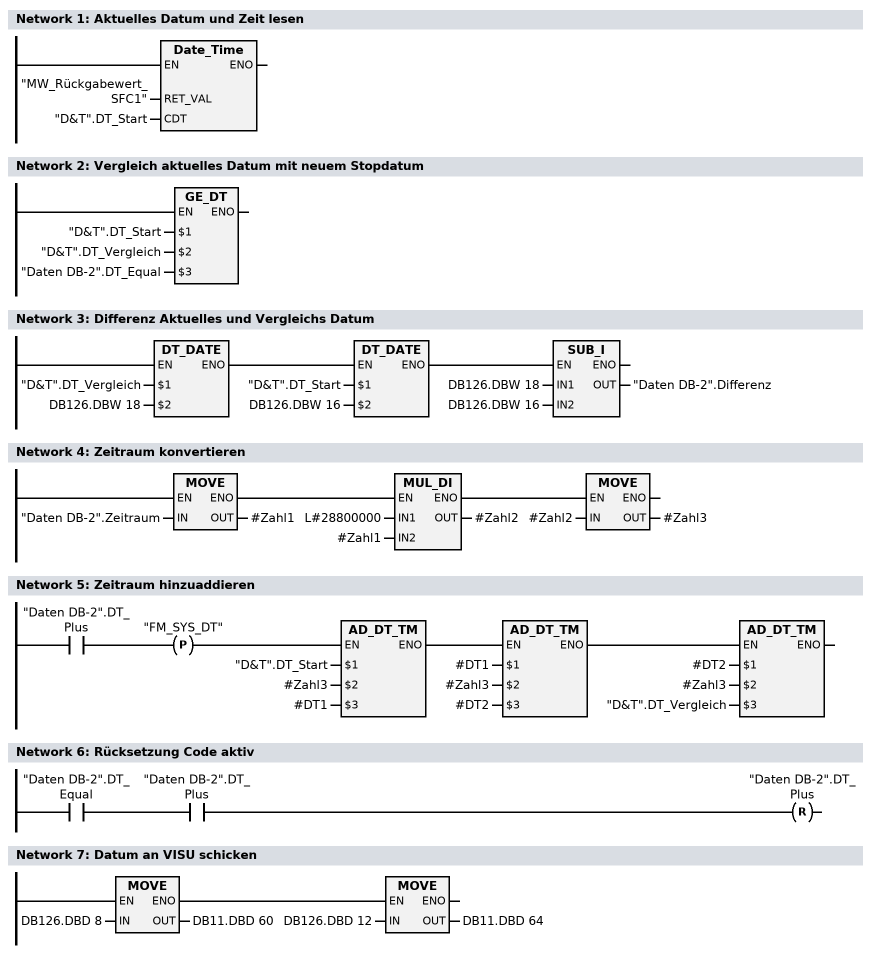
NETWORK
TITLE = Aktuelles Datum und Zeit lesen
      CALL  "Date_Time" (
           RET_VAL                  := "MW_Rückgabewert_SFC1",
           CDT                      := "D&T".DT_Start);
NETWORK
TITLE = Vergleich aktuelles Datum mit neuem Stopdatum
      CALL  "GE_DT" (
           $1                       := "D&T".DT_Start,
           $2                       := "D&T".DT_Vergleich,
           $3                       := "Daten DB-2".DT_Equal);
      NOP   0;
NETWORK
TITLE = Differenz Aktuelles und Vergleichs Datum
      A(;
      A(;
      CALL  "DT_DATE" (
           $1                       := "D&T".DT_Vergleich,
           $2                       := DB126.DBW 18);
      A     BR;
      );
      JNB   _001;
      CALL  "DT_DATE" (
           $1                       := "D&T".DT_Start,
           $2                       := DB126.DBW 16);
_001: A     BR;
      );
      JNB   _002;
      L     DB126.DBW 18;
      L     DB126.DBW 16;
      -I;
      T     "Daten DB-2".Differenz;
_002: NOP   0;
NETWORK
TITLE = Zeitraum konvertieren
      A(;
      A(;
      L     "Daten DB-2".Zeitraum;
      T     #Zahl1;
      SET;
      SAVE;
      CLR;
      A     BR;
      );
      JNB   _003;
      L     L#28800000;
      L     #Zahl1;
      *D;
      T     #Zahl2;
      AN    OV;
      SAVE;
      CLR;
_003: A     BR;
      );
      JNB   _004;
      L     #Zahl2;
      T     #Zahl3;
_004: NOP   0;
NETWORK
TITLE = Zeitraum hinzuaddieren
      A(;
      A(;
      A     "Daten DB-2".DT_Plus;
      FP    "FM_SYS_DT";
      JNB   _005;
      CALL  "AD_DT_TM" (
           $1                       := "D&T".DT_Start,
           $2                       := #Zahl3,
           $3                       := #DT1);
_005: A     BR;
      );
      JNB   _006;
      CALL  "AD_DT_TM" (
           $1                       := #DT1,
           $2                       := #Zahl3,
           $3                       := #DT2);
_006: A     BR;
      );
      JNB   _007;
      CALL  "AD_DT_TM" (
           $1                       := #DT2,
           $2                       := #Zahl3,
           $3                       := "D&T".DT_Vergleich);
_007: NOP   0;
NETWORK
TITLE = Rücksetzung Code aktiv
      A     "Daten DB-2".DT_Equal;
      A     "Daten DB-2".DT_Plus;
      R     "Daten DB-2".DT_Plus;
NETWORK
TITLE = Datum an VISU schicken
      A(;
      L     DB126.DBD 8;
      T     DB11.DBD 60;
      SET;
      SAVE;
      CLR;
      A     BR;
      );
      JNB   _008;
      L     DB126.DBD 12;
      T     DB11.DBD 64;
_008: NOP   0;
END_FUNCTION

// FC 127: know-how protected block, not included

// FC 128: know-how protected block, not included

// FC 129: know-how protected block, not included

// FC 130: know-how protected block, not included

FUNCTION "CutterSpeed-A4VG250" : VOID	// FC 140
TITLE = Volumenstromeinstellung für Schürfrad BKAG132kW/CSG355
AUTHOR : Simdon
FAMILY : Cutter
NAME : CutVol3
VERSION : 0.1
VAR_TEMP
  Ltr_200 : BOOL ;	//115 ltr/min
  Ltr_270 : BOOL ;	//270 ltr/min
  Ltr_max : BOOL ;	//max. Fördermenge
END_VAR
BEGIN
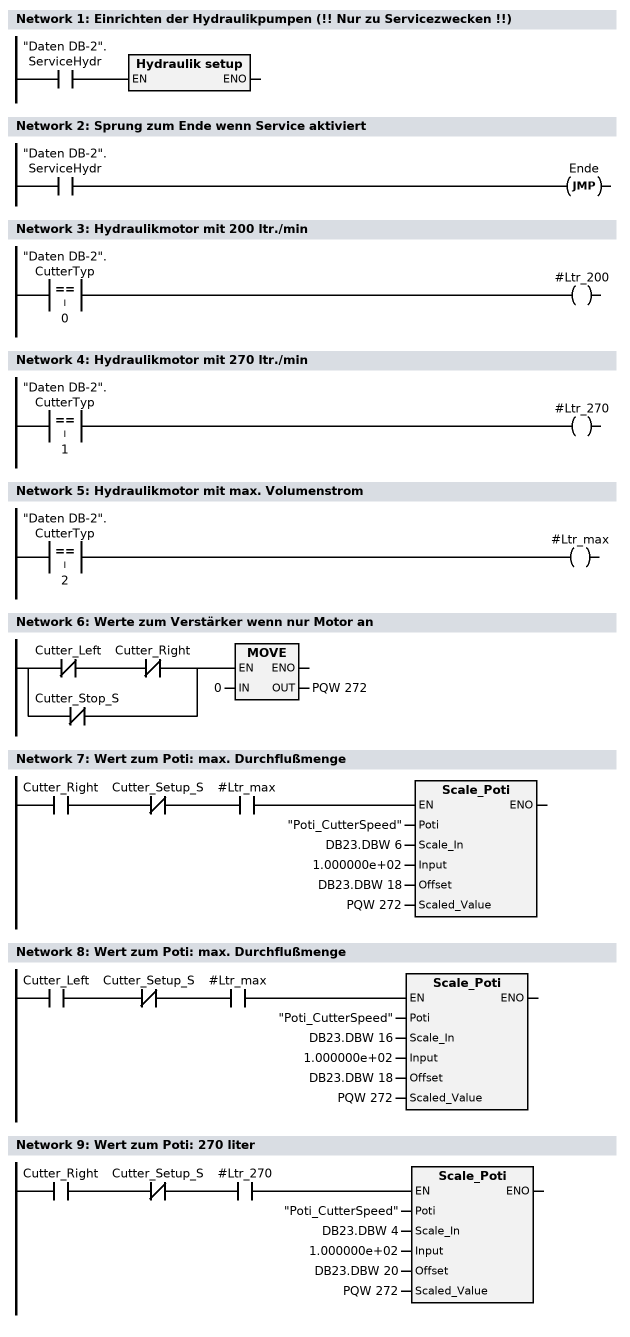
NETWORK
TITLE = Einrichten der Hydraulikpumpen (!! Nur zu Servicezwecken !!)
      A     "Daten DB-2".ServiceHydr;
      JNB   _001;
      CALL  "Hydraulik setup";
_001: NOP   0;
NETWORK
TITLE = Sprung zum Ende wenn Service aktiviert
      A     "Daten DB-2".ServiceHydr;
      JC    Ende;
NETWORK
TITLE = Hydraulikmotor mit 200 ltr./min
      L     "Daten DB-2".CutterTyp;
      L     0;
      ==I;
      =     #Ltr_200;
NETWORK
TITLE = Hydraulikmotor mit 270 ltr./min
      L     "Daten DB-2".CutterTyp;
      L     1;
      ==I;
      =     #Ltr_270;
NETWORK
TITLE = Hydraulikmotor mit max. Volumenstrom
      L     "Daten DB-2".CutterTyp;
      L     2;
      ==I;
      =     #Ltr_max;
NETWORK
TITLE = Werte zum Verstärker wenn nur Motor an
      A(;
      AN    "Cutter_Left";
      AN    "Cutter_Right";
      ON    "Cutter_Stop_S";
      );
      JNB   _002;
      L     0;
      T     PQW 272;
_002: NOP   0;
NETWORK
TITLE = Wert zum Poti: max. Durchflußmenge
      A     "Cutter_Right";
      AN    "Cutter_Setup_S";
      A     #Ltr_max;
      JNB   _003;
      CALL  "Scale_Poti" (
           Poti                     := "Poti_CutterSpeed",
           Scale_In                 := DB23.DBW 6,
           Input                    := 1.000000e+02,
           Offset                   := DB23.DBW 18,
           Scaled_Value             := PQW 272);
_003: NOP   0;
NETWORK
TITLE = Wert zum Poti: max. Durchflußmenge
      A     "Cutter_Left";
      AN    "Cutter_Setup_S";
      A     #Ltr_max;
      JNB   _004;
      CALL  "Scale_Poti" (
           Poti                     := "Poti_CutterSpeed",
           Scale_In                 := DB23.DBW 16,
           Input                    := 1.000000e+02,
           Offset                   := DB23.DBW 18,
           Scaled_Value             := PQW 272);
_004: NOP   0;
NETWORK
TITLE = Wert zum Poti: 270 liter
      A     "Cutter_Right";
      AN    "Cutter_Setup_S";
      A     #Ltr_270;
      JNB   _005;
      CALL  "Scale_Poti" (
           Poti                     := "Poti_CutterSpeed",
           Scale_In                 := DB23.DBW 4,
           Input                    := 1.000000e+02,
           Offset                   := DB23.DBW 20,
           Scaled_Value             := PQW 272);
_005: NOP   0;
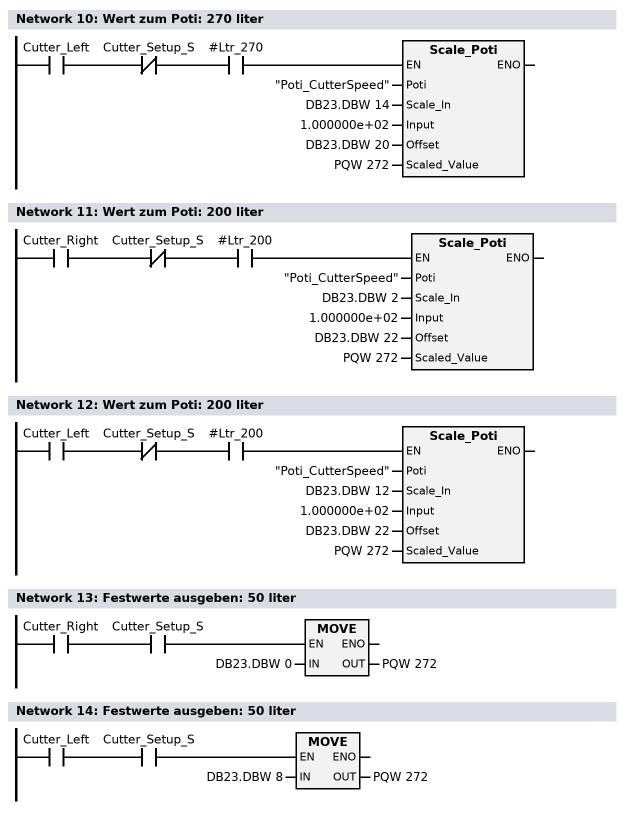
NETWORK
TITLE = Wert zum Poti: 270 liter
      A     "Cutter_Left";
      AN    "Cutter_Setup_S";
      A     #Ltr_270;
      JNB   _006;
      CALL  "Scale_Poti" (
           Poti                     := "Poti_CutterSpeed",
           Scale_In                 := DB23.DBW 14,
           Input                    := 1.000000e+02,
           Offset                   := DB23.DBW 20,
           Scaled_Value             := PQW 272);
_006: NOP   0;
NETWORK
TITLE = Wert zum Poti: 200 liter
      A     "Cutter_Right";
      AN    "Cutter_Setup_S";
      A     #Ltr_200;
      JNB   _007;
      CALL  "Scale_Poti" (
           Poti                     := "Poti_CutterSpeed",
           Scale_In                 := DB23.DBW 2,
           Input                    := 1.000000e+02,
           Offset                   := DB23.DBW 22,
           Scaled_Value             := PQW 272);
_007: NOP   0;
NETWORK
TITLE = Wert zum Poti: 200 liter
      A     "Cutter_Left";
      AN    "Cutter_Setup_S";
      A     #Ltr_200;
      JNB   _008;
      CALL  "Scale_Poti" (
           Poti                     := "Poti_CutterSpeed",
           Scale_In                 := DB23.DBW 12,
           Input                    := 1.000000e+02,
           Offset                   := DB23.DBW 22,
           Scaled_Value             := PQW 272);
_008: NOP   0;
NETWORK
TITLE = Festwerte ausgeben: 50 liter
      A     "Cutter_Right";
      A     "Cutter_Setup_S";
      JNB   _009;
      L     DB23.DBW 0;
      T     PQW 272;
_009: NOP   0;
NETWORK
TITLE = Festwerte ausgeben: 50 liter
      A     "Cutter_Left";
      A     "Cutter_Setup_S";
      JNB   _00a;
      L     DB23.DBW 8;
      T     PQW 272;
_00a: NOP   0;
NETWORK
TITLE = Bausteinende
Ende: NOP   0;
END_FUNCTION

FUNCTION "InterPresSpeed-A4VG250" : VOID	// FC 141
TITLE = Regelung für Dehner 4-6 (BKAG 132kW/A4VG250)
AUTHOR : Simdon
FAMILY : Presse
NAME : IntPresV
VERSION : 0.1
BEGIN
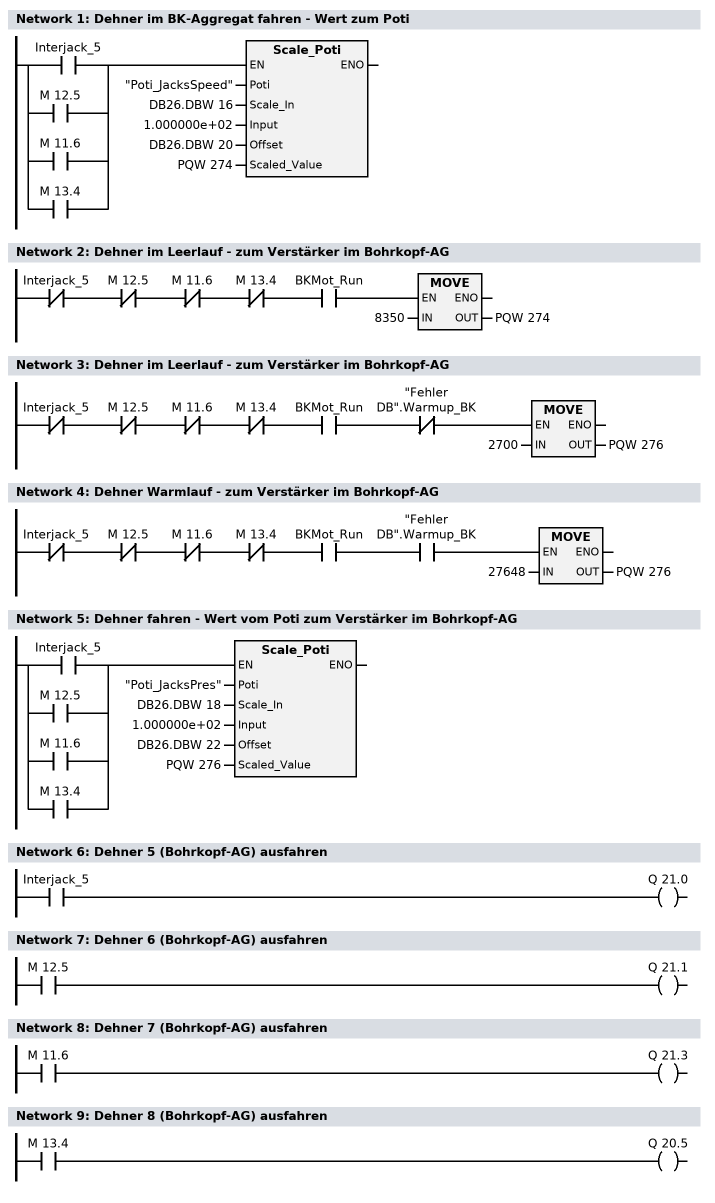
NETWORK
TITLE = Dehner im BK-Aggregat fahren - Wert zum Poti 
      A(;
      O     "Interjack_5";
      O     M 12.5;
      O     M 11.6;
      O     M 13.4;
      );
      JNB   _001;
      CALL  "Scale_Poti" (
           Poti                     := "Poti_JacksSpeed",
           Scale_In                 := DB26.DBW 16,
           Input                    := 1.000000e+02,
           Offset                   := DB26.DBW 20,
           Scaled_Value             := PQW 274);
_001: NOP   0;
NETWORK
TITLE = Dehner im Leerlauf - zum Verstärker im Bohrkopf-AG
      AN    "Interjack_5";
      AN    M 12.5;
      AN    M 11.6;
      AN    M 13.4;
      A     "BKMot_Run";
      JNB   _002;
      L     8350;
      T     PQW 274;
_002: NOP   0;
NETWORK
TITLE = Dehner im Leerlauf - zum Verstärker im Bohrkopf-AG
      AN    "Interjack_5";
      AN    M 12.5;
      AN    M 11.6;
      AN    M 13.4;
      A     "BKMot_Run";
      AN    "Fehler DB".Warmup_BK;
      JNB   _003;
      L     2700;
      T     PQW 276;
_003: NOP   0;
NETWORK
TITLE = Dehner Warmlauf - zum Verstärker im Bohrkopf-AG
      AN    "Interjack_5";
      AN    M 12.5;
      AN    M 11.6;
      AN    M 13.4;
      A     "BKMot_Run";
      A     "Fehler DB".Warmup_BK;
      JNB   _004;
      L     27648;
      T     PQW 276;
_004: NOP   0;
NETWORK
TITLE = Dehner fahren - Wert vom Poti zum Verstärker im Bohrkopf-AG
      A(;
      O     "Interjack_5";
      O     M 12.5;
      O     M 11.6;
      O     M 13.4;
      );
      JNB   _005;
      CALL  "Scale_Poti" (
           Poti                     := "Poti_JacksPres",
           Scale_In                 := DB26.DBW 18,
           Input                    := 1.000000e+02,
           Offset                   := DB26.DBW 22,
           Scaled_Value             := PQW 276);
_005: NOP   0;
NETWORK
TITLE = Dehner 5 (Bohrkopf-AG) ausfahren
      A     "Interjack_5";
      =     Q 21.0;
NETWORK
TITLE = Dehner 6 (Bohrkopf-AG) ausfahren 
      A     M 12.5;
      =     Q 21.1;
NETWORK
TITLE = Dehner 7 (Bohrkopf-AG) ausfahren 
      A     M 11.6;
      =     Q 21.3;
NETWORK
TITLE = Dehner 8 (Bohrkopf-AG) ausfahren 
      A     M 13.4;
      =     Q 20.5;
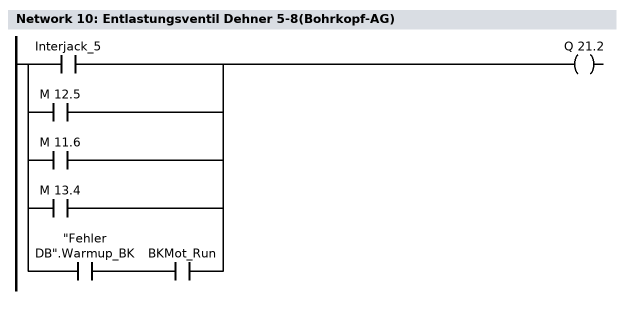
NETWORK
TITLE = Entlastungsventil Dehner 5-8(Bohrkopf-AG) 
      O     "Interjack_5";
      O     M 12.5;
      O     M 11.6;
      O     M 13.4;
      O;
      A     "Fehler DB".Warmup_BK;
      A     "BKMot_Run";
      =     Q 21.2;
END_FUNCTION

FUNCTION "QP_InterBK_A4VG" : VOID	// FC 142
TITLE = Durchflußwerte für BK-Dehner A4VG-Aggregat 132kW
AUTHOR : Simdon
FAMILY : Inter
NAME : QPInter
VERSION : 0.1
BEGIN
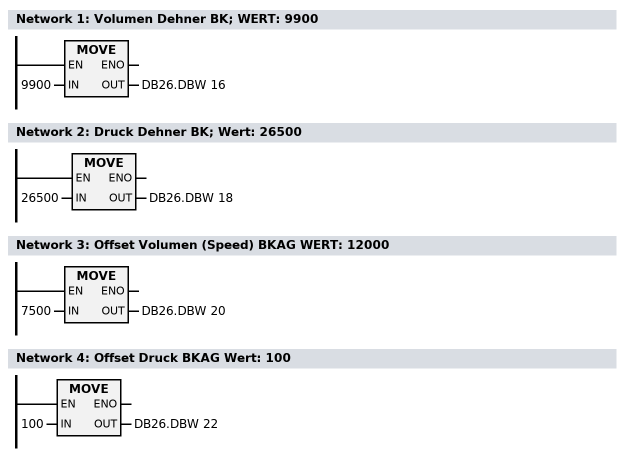
NETWORK
TITLE = Volumen Dehner BK; WERT: 9900
      L     9900;
      T     DB26.DBW 16;
      NOP   0;
NETWORK
TITLE = Druck Dehner BK; Wert: 26500
      L     26500;
      T     DB26.DBW 18;
      NOP   0;
NETWORK
TITLE = Offset Volumen (Speed) BKAG WERT: 12000
      L     7500;
      T     DB26.DBW 20;
      NOP   0;
NETWORK
TITLE = Offset Druck BKAG Wert: 100
      L     100;
      T     DB26.DBW 22;
      NOP   0;
END_FUNCTION

FUNCTION "CutterSpeed-CSG355" : VOID	// FC 150
TITLE = Volumenstromeinstellung für Schürfrad BKAG132kW/CSG355
AUTHOR : Simdon
FAMILY : Cutter
NAME : CutVol2
VERSION : 0.1
VAR_TEMP
  Ltr_200 : BOOL ;	//115 ltr/min
  Ltr_max : BOOL ;	//max. Fördermenge
  Ltr_270 : BOOL ;	//270 ltr/min
END_VAR
BEGIN
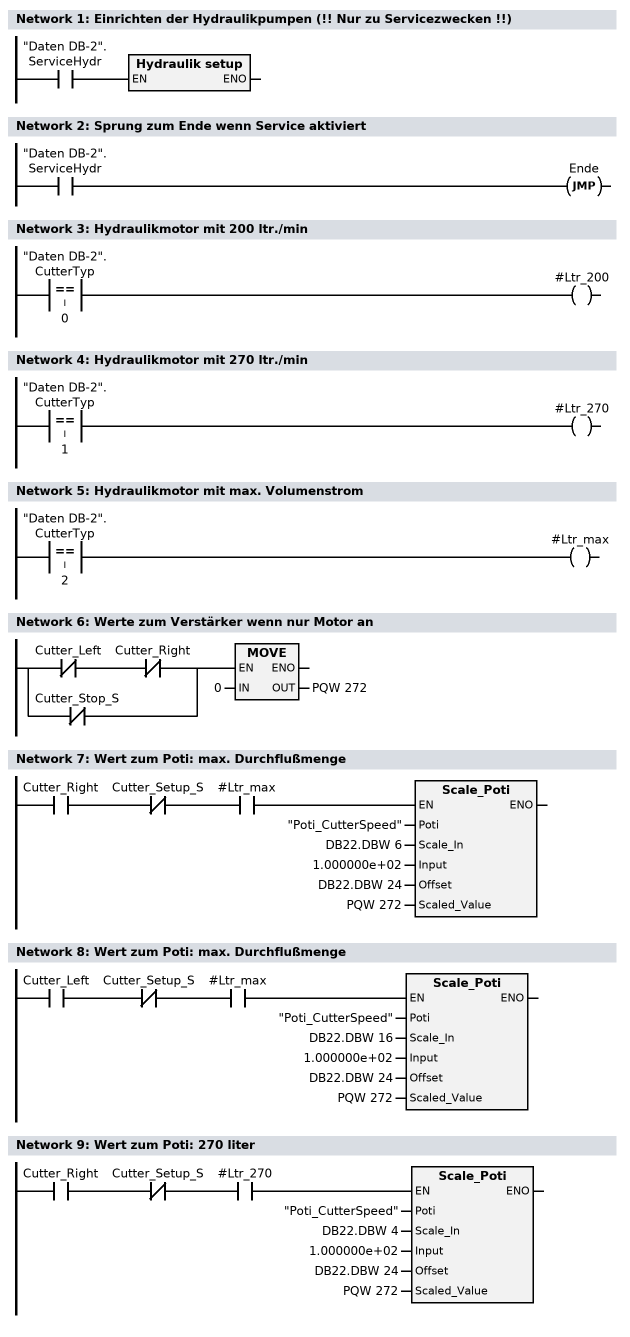
NETWORK
TITLE = Einrichten der Hydraulikpumpen (!! Nur zu Servicezwecken !!)
      A     "Daten DB-2".ServiceHydr;
      JNB   _001;
      CALL  "Hydraulik setup";
_001: NOP   0;
NETWORK
TITLE = Sprung zum Ende wenn Service aktiviert
      A     "Daten DB-2".ServiceHydr;
      JC    Ende;
NETWORK
TITLE = Hydraulikmotor mit 200 ltr./min
      L     "Daten DB-2".CutterTyp;
      L     0;
      ==I;
      =     #Ltr_200;
NETWORK
TITLE = Hydraulikmotor mit 270 ltr./min
      L     "Daten DB-2".CutterTyp;
      L     1;
      ==I;
      =     #Ltr_270;
NETWORK
TITLE = Hydraulikmotor mit max. Volumenstrom
      L     "Daten DB-2".CutterTyp;
      L     2;
      ==I;
      =     #Ltr_max;
NETWORK
TITLE = Werte zum Verstärker wenn nur Motor an
      A(;
      AN    "Cutter_Left";
      AN    "Cutter_Right";
      ON    "Cutter_Stop_S";
      );
      JNB   _002;
      L     0;
      T     PQW 272;
_002: NOP   0;
NETWORK
TITLE = Wert zum Poti: max. Durchflußmenge
      A     "Cutter_Right";
      AN    "Cutter_Setup_S";
      A     #Ltr_max;
      JNB   _003;
      CALL  "Scale_Poti" (
           Poti                     := "Poti_CutterSpeed",
           Scale_In                 := DB22.DBW 6,
           Input                    := 1.000000e+02,
           Offset                   := DB22.DBW 24,
           Scaled_Value             := PQW 272);
_003: NOP   0;
NETWORK
TITLE = Wert zum Poti: max. Durchflußmenge
      A     "Cutter_Left";
      AN    "Cutter_Setup_S";
      A     #Ltr_max;
      JNB   _004;
      CALL  "Scale_Poti" (
           Poti                     := "Poti_CutterSpeed",
           Scale_In                 := DB22.DBW 16,
           Input                    := 1.000000e+02,
           Offset                   := DB22.DBW 24,
           Scaled_Value             := PQW 272);
_004: NOP   0;
NETWORK
TITLE = Wert zum Poti: 270 liter
      A     "Cutter_Right";
      AN    "Cutter_Setup_S";
      A     #Ltr_270;
      JNB   _005;
      CALL  "Scale_Poti" (
           Poti                     := "Poti_CutterSpeed",
           Scale_In                 := DB22.DBW 4,
           Input                    := 1.000000e+02,
           Offset                   := DB22.DBW 24,
           Scaled_Value             := PQW 272);
_005: NOP   0;
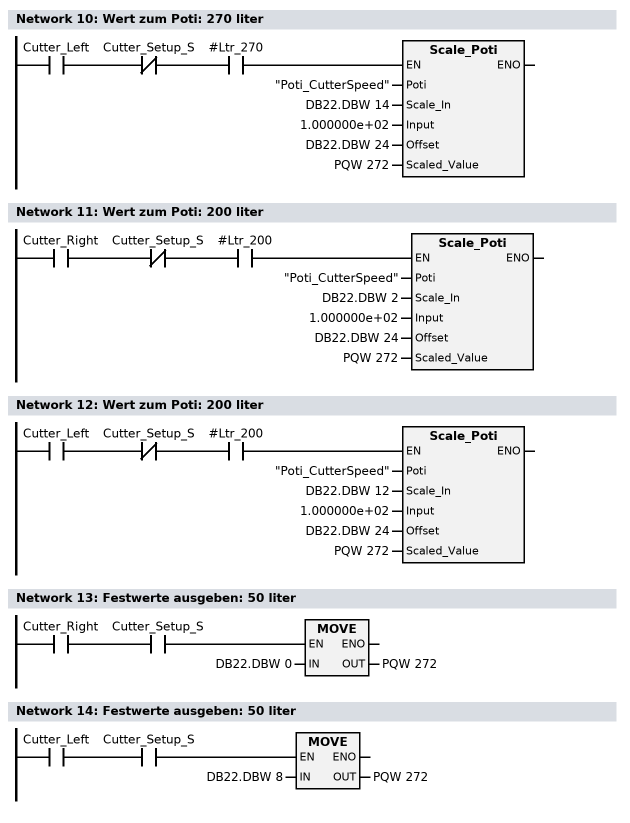
NETWORK
TITLE = Wert zum Poti: 270 liter
      A     "Cutter_Left";
      AN    "Cutter_Setup_S";
      A     #Ltr_270;
      JNB   _006;
      CALL  "Scale_Poti" (
           Poti                     := "Poti_CutterSpeed",
           Scale_In                 := DB22.DBW 14,
           Input                    := 1.000000e+02,
           Offset                   := DB22.DBW 24,
           Scaled_Value             := PQW 272);
_006: NOP   0;
NETWORK
TITLE = Wert zum Poti: 200 liter
      A     "Cutter_Right";
      AN    "Cutter_Setup_S";
      A     #Ltr_200;
      JNB   _007;
      CALL  "Scale_Poti" (
           Poti                     := "Poti_CutterSpeed",
           Scale_In                 := DB22.DBW 2,
           Input                    := 1.000000e+02,
           Offset                   := DB22.DBW 24,
           Scaled_Value             := PQW 272);
_007: NOP   0;
NETWORK
TITLE = Wert zum Poti: 200 liter
      A     "Cutter_Left";
      AN    "Cutter_Setup_S";
      A     #Ltr_200;
      JNB   _008;
      CALL  "Scale_Poti" (
           Poti                     := "Poti_CutterSpeed",
           Scale_In                 := DB22.DBW 12,
           Input                    := 1.000000e+02,
           Offset                   := DB22.DBW 24,
           Scaled_Value             := PQW 272);
_008: NOP   0;
NETWORK
TITLE = Festwerte ausgeben: 50 liter
      A     "Cutter_Right";
      A     "Cutter_Setup_S";
      JNB   _009;
      L     DB22.DBW 0;
      T     PQW 272;
_009: NOP   0;
NETWORK
TITLE = Festwerte ausgeben: 50 liter
      A     "Cutter_Left";
      A     "Cutter_Setup_S";
      JNB   _00a;
      L     DB22.DBW 8;
      T     PQW 272;
_00a: NOP   0;
NETWORK
TITLE = Bausteinende
Ende: NOP   0;
END_FUNCTION

FUNCTION "InterPresSpeed-CSG355" : VOID	// FC 151
TITLE = Volumenstrom und Druckregelung für Dehner 4-6 (BKAG 132kW/CSG35)
AUTHOR : Simdon
FAMILY : Presse
NAME : IntPresV
VERSION : 0.1
BEGIN
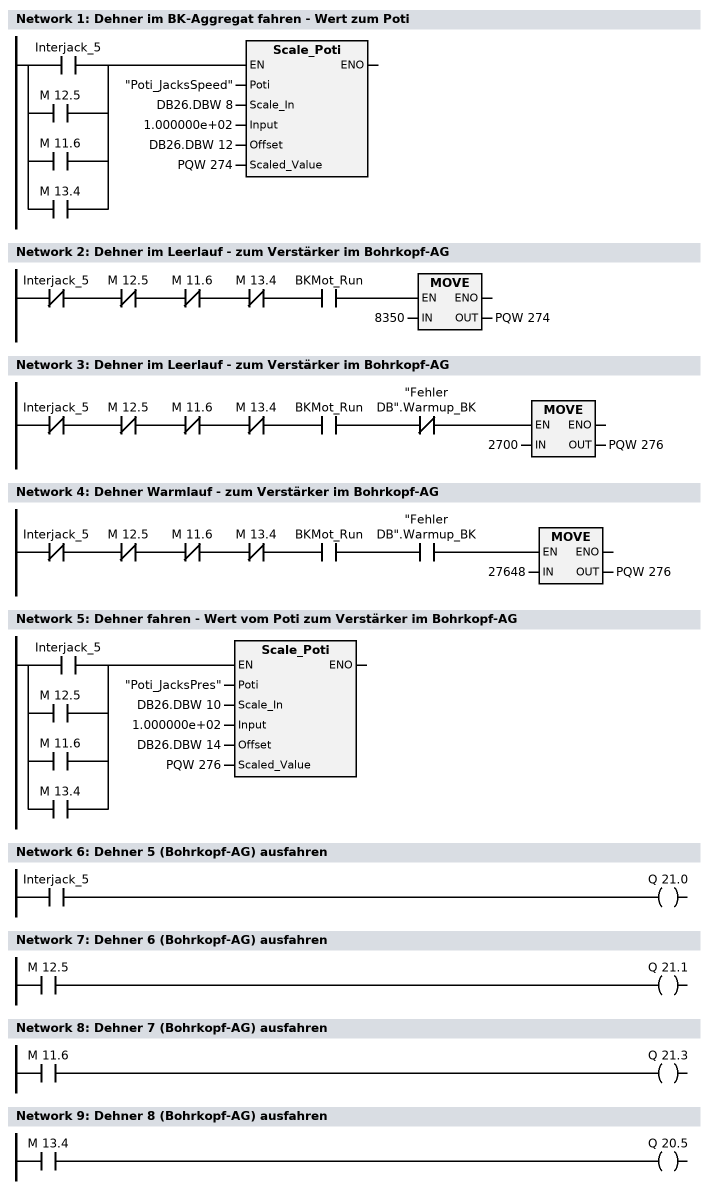
NETWORK
TITLE = Dehner im BK-Aggregat fahren - Wert zum Poti 
      A(;
      O     "Interjack_5";
      O     M 12.5;
      O     M 11.6;
      O     M 13.4;
      );
      JNB   _001;
      CALL  "Scale_Poti" (
           Poti                     := "Poti_JacksSpeed",
           Scale_In                 := DB26.DBW 8,
           Input                    := 1.000000e+02,
           Offset                   := DB26.DBW 12,
           Scaled_Value             := PQW 274);
_001: NOP   0;
NETWORK
TITLE = Dehner im Leerlauf - zum Verstärker im Bohrkopf-AG
      AN    "Interjack_5";
      AN    M 12.5;
      AN    M 11.6;
      AN    M 13.4;
      A     "BKMot_Run";
      JNB   _002;
      L     8350;
      T     PQW 274;
_002: NOP   0;
NETWORK
TITLE = Dehner im Leerlauf - zum Verstärker im Bohrkopf-AG
      AN    "Interjack_5";
      AN    M 12.5;
      AN    M 11.6;
      AN    M 13.4;
      A     "BKMot_Run";
      AN    "Fehler DB".Warmup_BK;
      JNB   _003;
      L     2700;
      T     PQW 276;
_003: NOP   0;
NETWORK
TITLE = Dehner Warmlauf - zum Verstärker im Bohrkopf-AG
      AN    "Interjack_5";
      AN    M 12.5;
      AN    M 11.6;
      AN    M 13.4;
      A     "BKMot_Run";
      A     "Fehler DB".Warmup_BK;
      JNB   _004;
      L     27648;
      T     PQW 276;
_004: NOP   0;
NETWORK
TITLE = Dehner fahren - Wert vom Poti zum Verstärker im Bohrkopf-AG
      A(;
      O     "Interjack_5";
      O     M 12.5;
      O     M 11.6;
      O     M 13.4;
      );
      JNB   _005;
      CALL  "Scale_Poti" (
           Poti                     := "Poti_JacksPres",
           Scale_In                 := DB26.DBW 10,
           Input                    := 1.000000e+02,
           Offset                   := DB26.DBW 14,
           Scaled_Value             := PQW 276);
_005: NOP   0;
NETWORK
TITLE = Dehner 5 (Bohrkopf-AG) ausfahren
      A     "Interjack_5";
      =     Q 21.0;
NETWORK
TITLE = Dehner 6 (Bohrkopf-AG) ausfahren 
      A     M 12.5;
      =     Q 21.1;
NETWORK
TITLE = Dehner 7 (Bohrkopf-AG) ausfahren 
      A     M 11.6;
      =     Q 21.3;
NETWORK
TITLE = Dehner 8 (Bohrkopf-AG) ausfahren 
      A     M 13.4;
      =     Q 20.5;
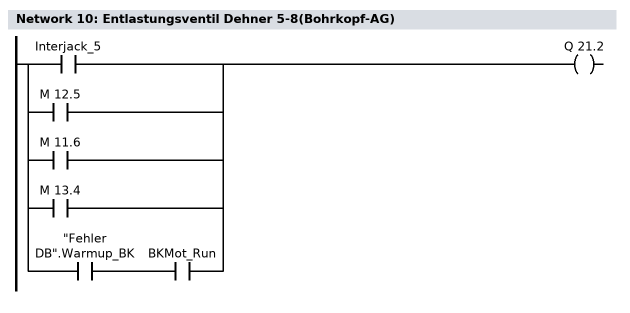
NETWORK
TITLE = Entlastungsventil Dehner 5-8(Bohrkopf-AG) 
      O     "Interjack_5";
      O     M 12.5;
      O     M 11.6;
      O     M 13.4;
      O;
      A     "Fehler DB".Warmup_BK;
      A     "BKMot_Run";
      =     Q 21.2;
END_FUNCTION

FUNCTION "QP_InterBK_CSG" : VOID	// FC 152
TITLE = Durchflußwerte für BK-Dehner CSG-Aggregat 132kW
AUTHOR : Simdon
FAMILY : Inter
NAME : QPInter
VERSION : 0.1
BEGIN
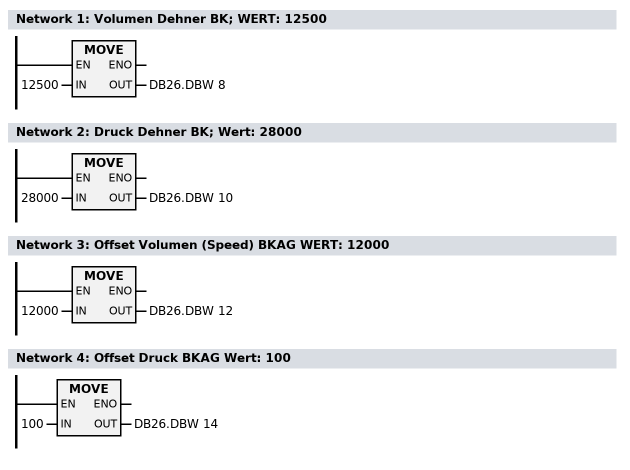
NETWORK
TITLE = Volumen Dehner BK; WERT: 12500
      L     12500;
      T     DB26.DBW 8;
      NOP   0;
NETWORK
TITLE = Druck Dehner BK; Wert: 28000
      L     28000;
      T     DB26.DBW 10;
      NOP   0;
NETWORK
TITLE = Offset Volumen (Speed) BKAG WERT: 12000
      L     12000;
      T     DB26.DBW 12;
      NOP   0;
NETWORK
TITLE = Offset Druck BKAG Wert: 100
      L     100;
      T     DB26.DBW 14;
      NOP   0;
END_FUNCTION

DATA_BLOCK "LV_DB"	// DB 1
AUTHOR : Simdon
FAMILY : LV
NAME : LV_DB
VERSION : 0.1
  STRUCT
   Zaehlwert : REAL ;	//vorläufige Platzhaltervariable
   T_Periode : REAL ;
   Speed : REAL ;
  END_STRUCT ;	
BEGIN
END_DATA_BLOCK

DATA_BLOCK "FU_DB1"	// DB 6
TITLE = Kontroll- und Rückgabewerte für FU´s und Softstarter
AUTHOR : Simdon
FAMILY : Motors
NAME : MOTDB1
VERSION : 0.1
  STRUCT
   BK_UmrichterStart : BOOL ;	//Ein 1 Signal schaltet den Umrichter ein
   BK_FReset : BOOL ;	//Eingang zum Rücksetzen einer Umrichterstörung
   BK_Alarm : BOOL ;	//Ausgang für Alarmmeldung vom Umrichter
   BK_UmrRun : BOOL ;	//Ausgang zeigt an ob der Umrichter läuft
   BK_UmrSSt : BOOL ;	//Bei 1 Signal liegt im Umrichter ein Fehler vor
   BK_KommSt : BOOL ;	//Kommunikationsstörung zum DP-Modul, bei NetzEin = 0 keine Auswertung
   C_UmrichterStart : BOOL ;	//Ein 1 Signal schaltet den Umrichter ein
   C_FReset : BOOL ;	//Eingang zum Rücksetzen einer Umrichterstörung
   C_Alarm : BOOL ;	//Ausgang für Alarmmeldung vom Umrichter
   C_UmrRun : BOOL ;	//Ausgang zeigt an ob der Umrichter läuft
   C_UmrSSt : BOOL ;	//Bei 1 Signal liegt im Umrichter ein Fehler vor
   C_KommSt : BOOL ;	//Kommunikationsstörung zum DP-Modul, bei NetzEin = 0 keine Auswertung
   D_NetzEin : BOOL ;	//Netzeingang, "1" Umrichter kann gestartet werden
   D_UmrichterStart : BOOL ;	//Ein 1 Signal schaltet den Umrichter ein
   D_FReset : BOOL ;	//Eingang zum Rücksetzen einer Umrichterstörung
   D_Alarm : BOOL ;	//Ausgang für Alarmmeldung vom Umrichter
   D_UmrRun : BOOL ;	//Ausgang zeigt an ob der Umrichter läuft
   D_UmrSSt : BOOL ;	//Bei 1 Signal liegt im Umrichter ein Fehler vor
   D_KommSt : BOOL ;	//Kommunikationsstörung zum DP-Modul, bei NetzEin = 0 keine Auswertung
   B_UmrichterStart : BOOL ;	//Ein 1 Signal schaltet den Umrichter ein
   B_FReset : BOOL ;	//Eingang zum Rücksetzen einer Umrichterstörung
   B_Alarm : BOOL ;	//Ausgang für Alarmmeldung vom Umrichter
   B_UmrRun : BOOL ;	//Ausgang zeigt an ob der Umrichter läuft
   B_UmrSSt : BOOL ;	//Bei 1 Signal liegt im Umrichter ein Fehler vor
   B_KommSt : BOOL ;	//Kommunikationsstörung zum DP-Modul, bei NetzEin = 0 keine Auswertung
   B2_UmrichterStart : BOOL ;	//Ein 1 Signal schaltet den Umrichter ein
   B2_FReset : BOOL ;	//Eingang zum Rücksetzen einer Umrichterstörung
   B2_Alarm : BOOL ;	//Ausgang für Alarmmeldung vom Umrichter
   B2_UmrRun : BOOL ;	//Ausgang zeigt an ob der Umrichter läuft
   B2_UmrSSt : BOOL ;	//Bei 1 Signal liegt im Umrichter ein Fehler vor
   B2_KommSt : BOOL ;	//Kommunikationsstörung zum DP-Modul, bei NetzEin = 0 keine Auswertung
   B3_NetzEin : BOOL ;	//Netzeingang, "1" Umrichter kann gestartet werden
   B3_UmrichterStart : BOOL ;	//Ein 1 Signal schaltet den Umrichter ein
   B3_FReset : BOOL ;	//Eingang zum Rücksetzen einer Umrichterstörung
   B3_Drehrichtung : BOOL ;	//Eingang für Dehrichtung
   B3_UmrRun : BOOL ;	//Ausgang zeigt an ob der Umrichter läuft
   B3_UmrSSt : BOOL ;	//Bei 1 Signal liegt im Umrichter ein Fehler vor
   B3_KommSt : BOOL ;	//Kommunikationsstörung zum DP-Modul, bei NetzEin = 0 keine Auswertung
   BK_DrzSoll : WORD ;	//Drehzahlsollwert für den Umrichter - Eingabe ohne Skalierung
   BK_MotorSpg : INT ;	//Istwert Motorspannung
   BK_NetzSpg : INT ;	//Istwert Netzspannung
   C_DrzSoll : WORD ;	//Drehzahlsollwert für den Umrichter - Eingabe ohne Skalierung
   C_MotorSpg : INT ;	//Istwert Motorspannung
   C_NetzSpg : INT ;	//Istwert Netzspannung
   D_DrzSoll : WORD ;	//Drehzahlsollwert für den Umrichter - Eingabe ohne Skalierung
   D_MotorSpg : INT ;
   D_NetzSpg : INT ;
   B_DrzSoll : WORD ;	//Drehzahlsollwert für den Umrichter - Eingabe ohne Skalierung
   B_MotorSpg : INT ;
   B_NetzSpg : INT ;
   B2_DrzSoll : WORD ;	//Drehzahlsollwert für den Umrichter - Eingabe ohne Skalierung
   B2_MotorSpg : INT ;
   B2_NetzSpg : INT ;
   B3_DrzSoll : WORD ;	//Drehzahlsollwert für den Umrichter - Eingabe ohne Skalierung
   B3_MotorSpg : INT ;
   B3_NetzSpg : INT ;
  END_STRUCT ;	
BEGIN
END_DATA_BLOCK

DATA_BLOCK "FU_DB2"	// DB 7
TITLE = Rückgabewerte der FU´s für Visualisierung
AUTHOR : Simdon
FAMILY : Motors
NAME : MOTDB2
VERSION : 0.1
  STRUCT
   BK_FNum : INT ;	//Fehlernummer des Umrichters
   BK_DrzIst : INT ;	//Bohrkopfmotor Drehzahlistwert
   BK_StromIst : INT ;	//Istwert Motorstrom
   BK_PowerIst : INT ;	//Prozent der Motorleistung
   BK_BetrStd : INT ;	//Gesamtanzahl der Betriebsstunden
   C_Fnum : INT ;	//Fehlernummer des Umrichters
   C_DrzIst : INT ;	//Drehzahlistwert des Umrichters - Ausgabe ohne Skalierung
   C_StromIst : INT ;	//Istwert Motorstrom
   C_PowerIst : INT ;	//Prozent der Motorleistung
   C_BetrStd : INT ;	//Betriebsstunden Motor
   D_Fnum : INT ;	//Fehlernummer des Umrichters
   D_DrzIst : INT ;	//Drehzahlistwert des Umrichters - Ausgabe ohne Skalierung
   D_StromIst : INT ;
   D_PowerIst : INT ;
   D_BetrStd : INT ;
   B_Fnum : INT ;	//Fehlernummer des Umrichters
   B_DrzIst : INT ;	//Drehzahlistwert des Umrichters - Ausgabe ohne Skalierung
   B_StromIst : INT ;
   B_PowerIst : INT ;
   B_BetrStd : INT ;
   B2_Fnum : INT ;	//Fehlernummer des Umrichters
   B2_DrzIst : INT ;	//Drehzahlistwert des Umrichters - Ausgabe ohne Skalierung
   B2_StromIst : INT ;
   B2_PowerIst : INT ;
   B2_BetrStd : INT ;
   B3_Fnum : INT ;	//Fehlernummer des Umrichters
   B3_DrzIst : INT ;	//Drehzahlistwert des Umrichters - Ausgabe ohne Skalierung
   B3_StromIst : INT ;
   B3_PowerIst : INT ;
   B3_BetrStd : INT ;
  END_STRUCT ;	
BEGIN
END_DATA_BLOCK

DATA_BLOCK "SO_DB1"	// DB 8
AUTHOR : Simdon
FAMILY : MotDB
NAME : SODB1
VERSION : 0.1
  STRUCT
   Ausgangsfrequenz : INT ;	//Ausgangsfrequenz 0..100Hz [0..200]
   Netzfrequenz : INT ;	//Netzfrequenz 0..100Hz [0..200]
   U_L1_L2 : INT ;	//Verkettete Spannung 0..1500V [0..15000]
   U_L2_L3 : INT ;	//Verkettete Spannung 0..1500V [0..15000]
   U_L3_L1 : INT ;	//Verkettete Spannung 0..1500V [0..15000]
   Strom_L1_Eff : REAL ;	//Phasenstrom L1 0..20 000 A [0..2 000 000]
   Strom_L2_Eff : REAL ;	//Phasenstrom L2 0..20 000 A [0..2 000 000]
   Strom_L3_Eff : REAL ;	//Phasenstrom L3 0..20 000 A [0..2 000 000]
   Ausgangsleistung : REAL ;	//Ausgangsleistung 0..2 147 483 W [0.. 2 147 4830]
  END_STRUCT ;	
BEGIN
END_DATA_BLOCK

DATA_BLOCK "Daten_DB"	// DB 10
TITLE = Werte für Visualisierung u. Protokollierung
AUTHOR : Simdon
NAME : PC_Daten
VERSION : 0.1
  STRUCT
   Cutter_RPM : REAL ;	//Drehzahl Schürfscheibe
   Cutter_Pressure : REAL ;	//Druck Schürfrad
   Jacks_Force : REAL ;	//Kraft Hauptpresse
   SlurryChamber_Pres : REAL ;	//Druck Spuelkammer
   SlurryLine_Pres : REAL ;	//Druck Spuelleitung
   Steering_Pres : REAL ;	//Druck Steuerung
   ChargeFlow : REAL ;	//Durchfluss Speiseleitung
   DischargeFlow : REAL ;	//Durchfluss Förderleitung
   VerticalDev : REAL ;	//Vertikale Abweichung
   HorizontalDev : REAL ;	//Horizontale Abweichung
   Headroll : REAL ;	//Verrollung von Zieltafel
   Gradient : REAL ;	//Längsneigung von Zieltafel
   Inclinometer : REAL ;	//Zusatz-Inklinometer
   DriveLength : REAL ;	//Vortriebslänge
   HydrOilTemp_Head : REAL ;	//Hydrauliköltemperatur im Bohrkopftank
   HydrOilTemp_PP : REAL ;	//Hydrauliköltemperatur im Containertank
   Cyl1_Way : REAL ;	//Wegaufnehmer Steuerzylinder 1
   Cyl2_Way : REAL ;	//Wegaufnehmer Steuerzylinder 2
   Cyl3_Way : REAL ;	//Wegaufnehmer Steuerzylinder 3
   Cyl1_Pres : REAL ;	//Druckaufnehmer Steuerzylinder 1
   Cyl2_Pres : REAL ;	//Druckaufnehmer Steuerzylinder 2
   Cyl3_Pres : REAL ;	//Druckaufnehmer Steuerzylinder 3
   Inter1_Way : REAL ;	//Wegaufnehmer Dehnerstation 1
   Inter2_Way : REAL ;	//Wegaufnehmer Dehnerstation 2
   Inter3_Way : REAL ;	//Wegaufnehmer Dehnerstation 3
   Inter4_Way : REAL ;	//Wegaufnehmer Dehnerstation 4
   Inter1_Pres : REAL ;	//Druckaufnehmer Dehnerstation 1
   Inter2_Pres : REAL ;	//Druckaufnehmer Dehnerstation 2
   Inter3_Pres : REAL ;	//Druckaufnehmer Dehnerstation 3
   Inter4_Pres : REAL ;	//Druckaufnehmer Dehnerstation 4
   Wing_Way : REAL ;	//Wegaufnehmer Flosse
   Crusher_Way : REAL ;	//Wegaufnehmer Brecher
   Charge_RPM : REAL ;	//Drehzahl Speisepumpe
   Discharge_RPM : REAL ;	//Drehzahl Förderpumpe
   Booster_RPM : REAL ;	//Drehzahl Zusatzpumpe
   DriveStatus : BOOL ;	//Status für den Vortrieb
   BypassOpen : BOOL ;	//Bypassventil ist geöffnet (Bypass)
   BypassClosed : BOOL ;	//Bypassventil ist geschlossen (Spülen)
   JetOpen : BOOL ;	//Jetventil ist geöffnet (Jet)
   JetClosed : BOOL ;	//Jetventil ist geöffnet (Spülen)
   Spare0 : BOOL ;
   Spare1 : BOOL ;
   Spare2 : BOOL ;
   BypassHeadroll : BOOL ;	//Überbrückung Verrollung
   BypassCaseDrain : BOOL ;	//Überbrückung Lecköl
   CaseDrain : BOOL ;	//Lecköldrucksensor
   GasAlarm : BOOL ;	//Sammelalarm der Gassensorik
   Spare8 : BOOL ;
   SafePosition : BOOL ;	//Stellung der Schürfscheibe okay
   JetBypass : BOOL ;	//Anzeige für Bypass-Spülen und Jet auf
   Prot_Activ : BOOL ;	//Protokollierung ist aktiv
   TACS_TargetInfo : WORD ;	//Infos vom Target: 0=Fehler, 5=Inclinometer Fail, 7=okay
   Spare10 : BOOL ;	//Steuerung der Datenprotokollierung
   Spare101 : BOOL ;
   Spare102 : BOOL ;
   Spare103 : BOOL ;
   Spare104 : BOOL ;
   Spare105 : BOOL ;
   Spare106 : BOOL ;
   Spare107 : BOOL ;
   Prot_Allgemein : BOOL ;	//Protokollbild für allgemeine Daten (1/72/0/1)
   Prot_HydrCont : BOOL ;	//Protokollbild für Daten Hydraulik-AG Container (1/72/1/1)
   Prot_Slurry : BOOL ;	//Protokollbild für Daten der Spülpumpen (1/72/2/1)
   Prot_HydrBKAG : BOOL ;	//Protokollbild für Daten Hydraulik Bohrkopf-AG (1/72/4/1)
   Prot_Service : BOOL ;	//Protokollbild für Daten Service/Setup (1/72/5/1)
   Richtungsabw : REAL ;
   SpeedJacks : REAL ;	//Vortriebsgeschwindigkeit
   RPMBooster2 : REAL ;	//Drehzahl Zusatzpumpe 2
   RPMBooster3 : REAL ;	//Drehzahl Zusatzpumpe 3
   Wing2_Way : REAL ;	//Wegaufnehmer Flosse 2
   Inter5_Way : REAL ;	//Wegaufnehmer Dehnerstation 5
   Inter5_Pres : REAL ;	//Druckaufnehmer Dehnerstation 5
   JacksPres : REAL ;	//Druckaufnehmer Hauptpresse
   MaxForceJacks : REAL ;	//Max. zugelassene Pressenkraft
   LockLeft : BOOL ;	//Verriegelungszylinder links verriegelt
   UnlockLeft : BOOL ;	//Verriegelungszylinder links entriegelt
   LockRight : BOOL ;	//Verriegelungszylinder rechts verriegelt
   UnlockRight : BOOL ;	//Verriegelungszylinder rechts entriegelt
   JacksRetracted : BOOL ;	//Druckbruecke hinten
   CutterLowRpm : BOOL ;	//Niedrige Drehzahl Cuter
   Frei6 : BOOL ;
   frei7 : BOOL ;
   MaxCutPres : REAL ;	//Max. zulässiger Schürfscheibendruck
   HD_Volume : REAL ;	//Volumenstrom Hochdruckwasserpumpe
   HD_Pressure : REAL ;	//Druck Hochdruckwasserpumpe
   Inter6_Way : REAL ;	//Wegaufnehmer Dehnerstation 6
   Inter6_Pres : REAL ;	//Druckaufnehmer Dehnerstation 6
   mtsNeigung : REAL ;
   JacksPres600 : REAL ;	//Druckaufnehmer Presse 500 bar Kreis
   AugerPres : REAL ;	//Druck Schneckenkreis
  END_STRUCT ;	
BEGIN
END_DATA_BLOCK

DATA_BLOCK "Daten DB-2"	// DB 11
TITLE = Einstellwerte für die Maschine
AUTHOR : Simdon
FAMILY : Dat_Log
NAME : PC_Daten
VERSION : 0.1
  STRUCT
   CylZeroAdj : BOOL ;	//Nullabgleich der Steuerzylinder
   JackingFrame : BOOL ;	//Auswahl der Hauptpresse (mts=1 oder HK=0)
   JacksActiv : BOOL ;	//Presse eingeschaltet
   T2 : BOOL ;
   DT_Equal : BOOL ;	//Vergleich aktuelles Datum mit neuem Stopdatum
   DT_Plus : BOOL ;	//Zeitraum hinzuaddieren
   DT_Start : BOOL ;	//Begin Zeitfenster für 1.Meldung
   CutterLeft : BOOL ;	//Anzeige für Schürfraddrehrichtung
   CutterRight : BOOL ;	//Anzeige für Schürfraddrehrichtung
   Crusher_Adj : BOOL ;	//Brecherverschiebung
   CorrectDistance : BOOL ;	//Korrektur der Vortriebslänge
   CutterMotorService : BOOL ;	//Schuerfradmotor starten ohne Wasserpumpe
   TimeProtocoll : BOOL ;	//Protokollierung über Zeitintervall
   ResetDistance : BOOL ;	//Zurücksetzen des Längenvortriebsgebers
   ReadBSCounter : BOOL ;	//Betriebsstundenzähler auslesen
   ServiceHydr : BOOL ;	//Service für Hydraulikpumpen
   BSCounterHydr : INT ;	//Betriebsstundenzähler für Hydraulikantrieb im Container-AG
   KorrekturDistance : REAL ;
   Lamptest : BOOL ;	//Lampentest für Pult
   InclZeroAdj : BOOL ;	//Nullabgleich vom Inclinometer (10/4/9/1)
   DN100 : BOOL ;	//Spülkreis DN 100 (10/4/10/1)
   DN125 : BOOL ;	//Spülkreis DN 125 (10/4/11/1)
   DN150 : BOOL ;	//Spülkreis DN 150 (10/4/12/1)
   DN200 : BOOL ;	//Spülkreis DN 200 (10/4/13/1)
   T16 : BOOL ;	//(10/4/14/1)
   Switch_mts1000 : BOOL ;	//Umschaltung auf mts1000(1); (10/4/15/1)
   Lock_Jet_Byp : BOOL ;	//Verriegelung von Jet und Bypass (0=Verriegelt, 1=Frei) (10/4/0/1)
   T18 : BOOL ;
   T19 : BOOL ;
   T20 : BOOL ;
   Gripper : BOOL ;	//Gripperstation eingebaut (Ja/Nein) (10/4/4/1)
   T22 : BOOL ;	//(10/4/5/1)
   Drive_Sim : BOOL ;	//Simulation für Status Vortrieb (10/4/6/1)
   Cooling_HydrOil : BOOL ;	//Externer Kühlkreis mit Pumpe für Hydrauliköl im Bohrkopf installiert (10/4/7/1)
   RPM_Faktor : REAL ;	//Faktor zur Drehzahlberechnung von der Visualisierung
   CylWay : INT ;	//Max. Hub der Steuerzylinder im Bohrkopf
   Inter1Way : REAL ;	//Max. Hub für Dehnerstation #1
   Inter2Way : REAL ;	//Max. Hub für Dehnerstation #2
   Inter3Way : REAL ;	//Max. Hub für Dehnerstation #3
   Inter4Way : REAL ;	//Max. Hub für Dehnerstation #4
   Inter5Way : REAL ;	//Max. Hub für Dehnerstation #5
   Inter6Way : REAL ;	//Max. Hub für Dehnerstation #6
   Slurrycircuit : INT ;	//Nennweite des Spülkreises
   CutterTyp : INT ;	//Auswahl für zulässige Literleistung beim Schürfradmotor (hydraulisch)
   RangeInclino : REAL ;
   Inter7Way : REAL ;	//Max. Hub für Dehnerstation #7
   Inter8Way : REAL ;	//Max. Hub für Dehnerstation #8
   Zeitraum : INT ;
   Differenz : INT ;
   SysDat : DATE_AND_TIME ;
   HD_Time : WORD ;	//Öffnungszeit für HD-Düsen/Ventile
  END_STRUCT ;	
BEGIN
END_DATA_BLOCK

DATA_BLOCK "Fehler DB"	// DB 13
TITLE = Fehlermeldungen von Sensoren, Füllstandsschaltern, etc.
AUTHOR : Simdon
FAMILY : System
NAME : Faults
VERSION : 0.1
  STRUCT
   Chargepump : BOOL ;	//Fehler Speisepumpe
   Dischargepump : BOOL ;	//Fehler Förderpumpe
   Boosterpump : BOOL ;	//Fehler Zusatzpumpe
   MainJackMot : BOOL ;	//Fehler Pressenmotor
   CutterMot : BOOL ;	//Fehler Schürfradmotor
   HydrOilFan1 : BOOL ;	//Fehler Hydrauliköllüfter #1
   HydrOilFan2 : BOOL ;	//Fehler Hydrauliköllüfter #2
   Steeringpump : BOOL ;	//Fehler Steuerpumpenmotor
   Booster2_Fault : BOOL ;	//Fehler Zusatzpumpe #2
   Booster3_Fault : BOOL ;	//Fehler Zusatzpumpe #3
   PreBypassFilte_PP : BOOL ;	//Voralarm Bypassfilter im Container-AG
   PreMainfilter1_PP : BOOL ;	//Voralarm Rücklauffilter #1 im Container-AG
   PreMainfilter2_PP : BOOL ;	//Voralarm Rücklauffilter #2 im Container-AG
   Oillevel_Med_PP : BOOL ;	//Ölstand im Container-AG auf "Mitte" -> Vorwarnung
   Oillevel_Low_PP : BOOL ;	//Ölstand im Container-AG auf "Leer" -> Abschaltung
   Bypassfilter_PP : BOOL ;	//Bypassfilter im Container-AG verstopft
   Mainfilter1_PP : BOOL ;	//Haupfilter #1 im Container-AG verstopft
   Mainfilter2_PP : BOOL ;	//Haupfilter #2 im Container-AG verstopft
   Warmup_PP : BOOL ;	//Hydrauliköltemperatur im Container-AG liegt unter 5°C
   Overheat_PP : BOOL ;	//Hydrauliköltemperatur im Container-AG liegt über 70°C
   Overheat2_PP : BOOL ;	//Hydrauliköltemperatur im Container-AG liegt über 90°C
   Oillevel_Med_BK : BOOL ;	//Ölstand im Bohrkopf-AG auf "Mitte" -> Vorwarnung
   Oillevel_Low_BK : BOOL ;	//Ölstand im Bohrkopf-AG auf "Leer" -> Abschaltung
   Returnlinefilter_BK : BOOL ;	//Rücklauffilter im Bohrkopfaggregat ist verstopft
   Warmup_BK : BOOL ;	//Hydrauliköltemperatur im Bohrkopf-AG liegt unter 5°C
   Overheat_BK : BOOL ;	//Hydrauliköltemperatur im Bohrkopf-AG liegt über 70°C
   Overheat2_BK : BOOL ;	//Hydrauliköltemperatur im Bohrkopf-AG liegt über 90°C
   FedCircuit_BK_low : BOOL ;	//Druck im Speisekreis ist zu niedrig
   FedCirFilter : BOOL ;	//Speisekreisfilter im BK-Aggregat ist verstopft
   CoolPump_EMotor : BOOL ;	//Zirkulationspumpe Kühlung E-Motor Bohrkopf ausgefallen
   CoolPump_HydrOil : BOOL ;	//Zirkulationspumpe Kühlung Hydrauliköl ausgefallen
   ThermoCutterMotor : BOOL ;	//Fehler Kaltleiter für den Bohrkopfmotor
   PreReturnlinefilter_BK : BOOL ;	//Voralarm Rücklauffilter im Bohrkopf-AG
   PreFedCirFilter_BK : BOOL ;	//Voralarm Speisekreisfilter im Bohrkopf-AG
   Cool_EMotor_BK : BOOL ;	//Durchflussmesser Kühlung E-Motor Bohrkopf < 40 l/min
   Cool_HydrOil_BK : BOOL ;	//Durchflussmesser Kühlkreislauf Hydrauliköl < 75 l/min
   RPM_Sensor_Fault : BOOL ;	//Ausfall Drehzahlsensor
   mts_Inclinometer : BOOL ;	//Fehler Zusatzinklinometer
   CaseDrain_high : BOOL ;	//Lecköldruck ist zu hoch
   Target_Roll : BOOL ;	//Verrollung ausserhalb des zulässigen Bereiches
   Target_Fault : BOOL ;	//Ausfall der Zieltafel
   TACSInclinometer : BOOL ;	//Verrollung der Zieltafel über 15° (links/rechts)
   NoLaser : BOOL ;	//Kein Laser auf dem Target
   LevelSw_Water_BK : BOOL ;	//Wasserstand im Bohrkopf ist zu hoch
   HD_Pump : BOOL ;	//Störung Hochdruckwasserpumpe
   FedCircuit_BKAG_low : BOOL ;	//Druck im Speisekreis BKKAG ist zu niedrig
   FedCirFilter_PP : BOOL ;	//Speisekreisfilter im PP-Aggregat ist verstopft
   PreFedCirFilter_PP : BOOL ;	//Voralarm Speisekreisfilter im PP-Aggregat
  END_STRUCT ;	
BEGIN
   Dischargepump := TRUE;
   Oillevel_Med_BK := TRUE;
   Oillevel_Low_BK := TRUE;
   Returnlinefilter_BK := TRUE;
   CaseDrain_high := TRUE;
   HD_Pump := TRUE;
   FedCirFilter_PP := TRUE;
END_DATA_BLOCK

DATA_BLOCK "Rückgabewerte"	// DB 14
TITLE = Rückgabewerte aus FC99, FC105, FC106, ...
AUTHOR : Simdon
FAMILY : Wandler
NAME : Return
VERSION : 0.1
  STRUCT
   Ret_Val_0 : WORD ;	//Rückgabewert
   Ret_Val_2 : WORD ;	//Rückgabewert
   Ret_Val_4 : WORD ;	//Rückgabewert
   Ret_Val_6 : WORD ;	//Rückgabewert
   Ret_Val_8 : WORD ;	//Rückgabewert
   Ret_Val_10 : WORD ;	//Rückgabewert
   Ret_Val_12 : WORD ;	//Rückgabewert
   Ret_Val_14 : WORD ;	//Rückgabewert
   Ret_Val_16 : WORD ;	//Rückgabewert
   Ret_Val_18 : WORD ;	//Rückgabewert
   Ret_Val_20 : WORD ;	//Rückgabewert
   Ret_Val_22 : WORD ;	//Rückgabewert
   Ret_Val_24 : WORD ;	//Rückgabewert
   Ret_Val_26 : WORD ;	//Rückgabewert
   Ret_Val_28 : WORD ;	//Rückgabewert
   Ret_Val_30 : WORD ;	//Rückgabewert
   Ret_Val_32 : WORD ;	//Rückgabewert
   Ret_Val_34 : WORD ;	//Rückgabewert
   Ret_Val_36 : WORD ;	//Rückgabewert
   Ret_Val_38 : WORD ;	//Rückgabewert
   Ret_Val_40 : WORD ;	//Rückgabewert
   Ret_Val_42 : WORD ;	//Rückgabewert
   Ret_Val_44 : WORD ;	//Rückgabewert
   Ret_Val_46 : WORD ;	//Rückgabewert
   Ret_Val_48 : WORD ;	//Rückgabewert
   Ret_Val_50 : WORD ;	//Rückgabewert
   Ret_Val_52 : WORD ;	//Rückgabewert
   Ret_Val_54 : WORD ;	//Rückgabewert
   Ret_Val_56 : WORD ;	//Rückgabewert
   Ret_Val_58 : WORD ;	//Rückgabewert
   Ret_Val_60 : WORD ;	//Rückgabewert
   Ret_Val_62 : WORD ;	//Rückgabewert
   Ret_Val_64 : WORD ;	//Rückgabewert
   Ret_Val_66 : WORD ;	//Rückgabewert
   Ret_Val_68 : WORD ;	//Rückgabewert
   Ret_Val_70 : WORD ;	//Rückgabewert
   Ret_Val_72 : WORD ;	//Rückgabewert
   Ret_Val_74 : WORD ;	//Rückgabewert
   Ret_Val_76 : WORD ;	//Rückgabewert
   Ret_Val_78 : WORD ;	//Rückgabewert
   Ret_Val_80 : WORD ;	//Rückgabewert
   ChargeStaus : INT ;	//Rückgabewert Charge
   DischargeStatus : INT ;	//Rückgabewert Discharge
  END_STRUCT ;	
BEGIN
END_DATA_BLOCK

DATA_BLOCK "Diverses"	// DB 15
AUTHOR : Simdon
FAMILY : Div
NAME : Diverses
VERSION : 0.1
  STRUCT
   ChargeFlow : REAL ;
   ChargeStatus : BYTE ;
   DischargeFlow : REAL ;
   DisStatus : BYTE ;
   Weg1 : REAL ;	//Zwischenwert für Geschwindigkeitsberechnung
   Weg2 : REAL ;	//Zwischenwert für Geschwindigkeitsberechnung
   Weg3 : REAL ;	//Zwischenwert für Geschwindigkeitsberechnung
   Weg4 : REAL ;	//Zwischenwert für Geschwindigkeitsberechnung
   Jacks_Adv : REAL ;	//Umrechnungsfaktor Bar-Tonnen
   Jacks_Ret : REAL ;	//Umrechnungsfaktor Bar-Tonnen
   Dehner : REAL ;	//Umrechnungsfaktor Bar-Tonnen
   Charge2 : REAL ;
   Charge2St : BYTE ;
   Discharge2 : REAL ;
   Discharge2St : BYTE ;
   RPM_In_Stat : BYTE ;	//Statusbyte für Piconet-Counter
   RPM_In_Dat1 : BYTE ;	//Input-Datenbyte 1
   RPM_In_Dat2 : BYTE ;	//Input-Datenbyte 2
   RPM_In_Dat3 : BYTE ;	//Input-Datenbyte 3
   RPM_In_Dat4 : BYTE ;	//Input-Datenbyte 4
   RPM_Out_Cont : BYTE ;	//Controlbyte für Piconet-Counter
   RPM_Out1 : BYTE ;	//Output-Datenbyte 1
   RPM_Out2 : BYTE ;	//Output-Datenbyte 2
   RPM_Out3 : BYTE ;	//Output-Datenbyte 3
   RPM_Out4 : BYTE ;	//Output-Datenbyte 4
   RPM_1 : REAL ;	//Zwischenwerte zur Drehzahlberchnung
   RPM_2 : REAL ;	//Zwischenwerte zur Drehzahlberchnung
   RPM_3 : REAL ;	//Zwischenwerte zur Drehzahlberchnung
   Weg_Speicher : REAL ;	//Gespeicherter Weg Haltung
   KraftDehnerBK : REAL ;	//Kraft der Dehner aus dem BK-Aggregat
   Weg_In_Stat1 : BYTE ;
   Weg_In_Stat2 : BYTE ;
   Weg_In_Stat3 : BYTE ;
   Weg_In_Stat4 : BYTE ;
   Weg_In_Data : DINT ;
   Weg_Out_Stat1 : BYTE ;
   Weg_Out_Stat2 : BYTE ;
   Weg_Out_Stat3 : BYTE ;
   Weg_Out_Stat4 : BYTE ;
   Weg_Out_Data : DINT ;
   Weg_Status : INT ;
   Inter_BK : REAL ;
   HD_Open : S5TIME ;	//Öffnungszeit der HD-Ventile
  END_STRUCT ;	
BEGIN
   ChargeFlow := -4.231780e-35;
   ChargeStatus := B#16#9C;
   DischargeFlow := -4.231780e-35;
   DisStatus := B#16#9C;
   Jacks_Adv := 1.212843e+00;
   Jacks_Ret := 2.463008e+00;
   Dehner := 3.302598e+00;
END_DATA_BLOCK

DATA_BLOCK "Analogvalues"	// DB 16
TITLE = Rückgabewerte von verschiedenen Sensoren und Poti´s
AUTHOR : Simdon
FAMILY : Control
NAME : Analog
VERSION : 0.1
  STRUCT
   JacksSpeed : REAL ;	//Rückgabewert vom Poti
   JacksPres : REAL ;	//Rückgabewert vom Poti
   CutterSpeed : REAL ;	//Rückgabewert vom Poti
   Zyl1_nlow : REAL ;	//Neue Untergrenze Wegaufnehmer Steuerzylinder 1
   Zyl1_nhigh : REAL ;	//Neue Obergrenze Wegaufnehmer Steuerzylinder 1
   Zyl2_nlow : REAL ;	//Neue Untergrenze Wegaufnehmer Steuerzylinder 2
   Zyl2_nhigh : REAL ;	//Neue Obergrenze Wegaufnehmer Steuerzylinder 2
   Zyl3_nlow : REAL ;	//Neue Untergrenze Wegaufnehmer Steuerzylinder 3
   Zyl3_nhigh : REAL ;	//Neue Obergrenze Wegaufnehmer Steuerzylinder 4
   Wing_nlow : REAL ;	//Neue Untergrenze Wegaufnehmer Flossenzylinder
   Wing_nhigh : REAL ;	//Neue Obergrenze Wegaufnehmer Flossenzylinder
   Pres_GreasePump : REAL ;	//Druck der Fettpumpe
   Inclino_mts_nlow : REAL ;	//Neuer Unterer Wert vom Inclinometer mts
   Inclino_mts_nhigh : REAL ;	//Neuer Oberer Wert vom Inclinometer mts
   Neigung_mts_nlow : REAL ;	//Neuer Unterer Wert vom Inclinometer (Neigung) mts
   Neigung_mts_nhigh : REAL ;	//Neuer Oberer Wert vom Inclinometer (Neigung) mts
  END_STRUCT ;	
BEGIN
END_DATA_BLOCK

DATA_BLOCK "Druck-Tonnen"	// DB 17
AUTHOR : Simdon
FAMILY : Jacks
NAME : P_zu_To
VERSION : 0.1
  STRUCT
   Jacks_Adv : REAL ;	//Umrechnungsfaktor Bar-Tonnen
   Jacks_Ret : REAL ;	//Umrechnungsfaktor Bar-Tonnen
   Dehner_1 : REAL ;	//Umrechnungsfaktor Bar-Tonnen
   Dehner_2 : REAL ;	//Umrechnungsfaktor Bar-Tonnen
   Dehner_3 : REAL ;	//Umrechnungsfaktor Bar-Tonnen
   Dehner_4 : REAL ;	//Umrechnungsfaktor Bar-Tonnen
   Dehner_5 : REAL ;	//Umrechnungsfaktor Bar-Tonnen
   Dehner_6 : REAL ;	//Umrechnungsfaktor Bar-Tonnen
   Dehner_7 : REAL ;	//Umrechnungsfaktor Bar-Tonnen
   Dehner_8 : REAL ;	//Umrechnungsfaktor Bar-Tonnen
  END_STRUCT ;	
BEGIN
END_DATA_BLOCK

DATA_BLOCK "Touchscreen"	// DB 19
TITLE = Aufnehmen und Weiterleiten der Werte für den Touchscreen
AUTHOR : Simdon
FAMILY : Visu
NAME : TS
VERSION : 0.1
  STRUCT
   Dehner_3 : BOOL ;	//Dehner 3 Ein/Ausschalten
   Dehner_4 : BOOL ;	//Dehner 4 Ein/Ausschalten
   Dehner_5 : BOOL ;	//Dehner 5 Ein/Ausschalten
   Brecher_Vor : BOOL ;	//Brecherverschiebung vorfahren
   Brecher_Zur : BOOL ;	//Brecherverschiebung zurückfahren
   RB_Set : BOOL ;	//Rohrbremse spannen
   RB_Rel : BOOL ;	//Rohrbremse lösen
   Bento_Valve_BK : BOOL ;	//Bentonitventil im Bohrkopf
   S_HD_Valve_1 : BOOL ;	//HD-Düse 1 ausgewählt
   S_HD_Valve_2 : BOOL ;	//HD-Düse 2 ausgewählt
   Roll_li : BOOL ;	//Überbrückung Verrollung links
   Roll_re : BOOL ;	//Überbrückung Verrollung rechts
   Leckoel : BOOL ;	//Überbrückung Lecköl
   Steuerung : BOOL ;	//Ventil Steuerung Ein/Ausschalten
   Dehner_1 : BOOL ;	//Dehner 1 Ein/Ausschalten
   Dehner_2 : BOOL ;	//Dehner 2 Ein/Ausschalten
   Dehner_8 : BOOL ;	//Dehner 8 Ein/Ausschalten
   HD_Pumpe : BOOL ;	//Hochdruckwasserpumpe Ein/Ausschalten
   Dehner_6 : BOOL ;	//Dehner 6 Ein/Ausschalten
   Dehner_7 : BOOL ;	//Dehner 7 Ein/Ausschalten
   HydrOilHead : BOOL ;	//Rohrbündelwärmetauscher Bohrkopfaggregat
   HD_Valve_Man : BOOL ;	//Manuelles Einschalten der HD-Ventile, keine HD-Pumpe mit SPS
   S_HD_Valve_3 : BOOL ;	//HD-Düse 3 ausgewählt
   S_HD_Valve_4 : BOOL ;	//HD-Düse 4 ausgewählt
   VerbZy_NL_vor : BOOL ;	//Verbindungszylinder im NL ausfahren
   VerbZy_NL_zur : BOOL ;	//Verbindungszylinder im NL einfahren
   BKLampe_1 : BOOL ;	//Lampe im Bohrkopf Ein/Ausschalten
   BKLampe_2 : BOOL ;	//Lampe im Nachläufer Ein/Ausschalten
   VerbZy_BK_vor : BOOL ;	//Verbindungszylinder im BK ausfahren
   VerbZy_BK_zur : BOOL ;	//Verbindungszylinder im BK einfahren
   Cam2_BK : BOOL ;	//Umschalten auf Kamera 2 (Rohr/Bohrkopf)
   S_HD_Auto : BOOL ;	//HD-Bedüsung im Automatikbetrieb
   Freigabe_Remote : BOOL ;	//Freigabe für Fernbedienung Presse
   Reserve_T1_1 : BOOL ;
   Reserve_T1_2 : BOOL ;
   Reserve_T1_3 : BOOL ;
   Reserve_T1_4 : BOOL ;
   Reserve_T1_5 : BOOL ;
   Reserve_T1_6 : BOOL ;
   Reserve_T1_7 : BOOL ;
   Reserve_T1_8_15 : BYTE ;
   Reserve_T_2 : WORD ;
   H_Dehner_3 : BOOL ;	//Dehner 3 eingeschaltet
   H_Dehner_4 : BOOL ;	//Dehner 4 eingeschaltet
   H_Dehner_5 : BOOL ;	//Dehner 5 eingeschaltet
   H_HD_Pumpe : BOOL ;	//Hochdruckwasserpumpe eingeschaltet
   H_Dehner_6 : BOOL ;	//Dehner 6 eingeschaltet
   H_HydrOilHead : BOOL ;	//Rohrbündelwärmetauscher Bohrkopfaggregat eingeschaltet
   H_LS_HD_Valve3 : BOOL ;	//Rückmeldung HD-Ventil 3 offen
   H_LS_HD_Valve4 : BOOL ;	//Rückmeldung HD-Ventil 4 offen
   H_LS_HD_Valve1 : BOOL ;	//Rückmeldung HD-Ventil 1 offen
   H_LS_HD_Valve2 : BOOL ;	//Rückmeldung HD-Ventil 2 offen
   H_Roll_li : BOOL ;	//Verrollung links
   H_Roll_re : BOOL ;	//Verrollung rechts
   H_Leckoel : BOOL ;	//Lecköl
   H_Steuerung : BOOL ;	//Steuerung
   H_Dehner_1 : BOOL ;	//Dehner 1 eingeschaltet
   H_Dehner_2 : BOOL ;	//Dehner 2 eingeschaltet
   H_Dehner_7 : BOOL ;	//Dehner 7 eingeschaltet
   H_Dehner_8 : BOOL ;	//Dehner 8 eingeschaltet
   Reserve_H_2 : WORD ;
  END_STRUCT ;	
BEGIN
END_DATA_BLOCK

DATA_BLOCK "Speed-Pres Jacks"	// DB 20
AUTHOR : Simdon
FAMILY : Presse
NAME : VolPres
VERSION : 0.1
  STRUCT
   V_6_Liter : INT ;	//Volumenstrom 6 l/min Verstärker
   V_50_Liter : INT ;	//Volumenstrom 50 l/min Verstärker
   V_136_Liter : INT ;	//Volumenstrom 136 l/min Verstärker, über Poti
   P_50_bar : INT ;	//Druck 50 bar
   P_100_bar : INT ;	//Druck 100 bar
   P_300_bar : INT ;	//Druck 300 bar; über Poti
   Offset_V : INT ;	//Offset für Poti Presse Geschwindigkeit
   Offset_P : INT ;	//Offset für Poti Presse Druck/Kraft
  END_STRUCT ;	
BEGIN
   V_50_Liter := 10250;
   V_136_Liter := 27648;
   P_50_bar := 4300;
   P_100_bar := 9000;
   P_300_bar := 25400;
END_DATA_BLOCK

DATA_BLOCK "Speed Cutter"	// DB 21
AUTHOR : Simdon
FAMILY : CutterAG
NAME : VolCut
VERSION : 0.1
  STRUCT
   V_50L_Rechts : INT ;	//Volumenstrom 50 l/min Rechts
   V_200L_Rechts : INT ;	//Volumenstrom 200 l/min Rechts
   V_270L_Rechts : INT ;	//Volumenstrom 270 l/min Rechts
   V_359L_Rechts : INT ;	//Volumenstrom 359 l/min Rechts
   V_50L_Links : INT ;	//Volumenstrom 50 l/min Links
   V_75L_Links : INT ;	//Volumenstrom 75 l/min Links
   V_200L_Links : INT ;	//Volumenstrom 200 l/min Links
   V_270L_Links : INT ;	//Volumenstrom 270 l/min Links
   V_359L_Links : INT ;	//Volumenstrom 359 l/min Links
   Offset_359L : INT ;	//Offset Cutter Speed 359 l/min
   Offset_270L : INT ;	//Offset Cutter Speed 270 l/min
   Offset_200L : INT ;	//Offset Cutter Speed 200 l/min
  END_STRUCT ;	
BEGIN
   V_50L_Rechts := 2150;
   V_200L_Rechts := 4500;
   V_270L_Rechts := 9800;
   V_359L_Rechts := 23500;
   V_50L_Links := -2150;
   V_75L_Links := -2900;
   V_200L_Links := -4500;
   V_270L_Links := -9800;
   V_359L_Links := -23500;
END_DATA_BLOCK

DATA_BLOCK "SO_DB2"	// DB 25
AUTHOR : Simdon
FAMILY : MotDB
NAME : SO_DB2
VERSION : 0.1
  STRUCT
   Strom_L1_Prozent : BYTE ;	//Phasenstrom L1 in %
   Strom_L2_Prozent : BYTE ;	//Phasenstrom L2 in %
   Strom_L3_Prozent : BYTE ;	//Phasenstrom L3 in %
   Reserviert_1 : BYTE ;
   Kuehlzeit_Motor : BYTE ;	//Verbleibende Abkülzeit des Motors
   Kuehlzeit_Motor1 : BYTE ;
   Motorwaerme : BYTE ;	//Motorwärme in %
   Unsymmetrie_40 : BYTE ;	//Bei Unsymmetrie > 40% = 1
   Unsymmetrie : BYTE ;	//Unsymmetrie in %
   Reserviert_2 : BYTE ;
   Reserviert_3 : BYTE ;
   Reserviert_4 : BYTE ;
   Reserviert_5 : BYTE ;
   Reserviert_6 : BYTE ;
   Reserviert_7 : BYTE ;
   Reserviert_8 : BYTE ;
   Ausgangsfrequenz : BYTE ;	//Ausgangsfrequenz 0..100Hz [0..200]
   Reserviert_9 : BYTE ;
   Reserviert_10 : BYTE ;
   Reserviert_11 : BYTE ;
   Netzfrequenz : BYTE ;	//Netzfrequenz 0..100Hz [0..200]
   Reserviert_12 : BYTE ;
   U_L1_L2 : BYTE ;	//Verkettete Spannung 0..1500V [0..15000]
   U_L1_L21 : BYTE ;
   U_L2_L3 : BYTE ;	//Verkettete Spannung 0..1500V [0..15000]
   U_L2_L31 : BYTE ;
   U_L3_L1 : BYTE ;	//Verkettete Spannung 0..1500V [0..15000]
   U_L3_L11 : BYTE ;
   Strom_L1_Eff : BYTE ;	//Phasenstrom L1 0..20 000 A [0..2 000 000]
   Strom_L1_Eff1 : BYTE ;
   Strom_L1_Eff2 : BYTE ;
   Strom_L1_Eff3 : BYTE ;
   Strom_L2_Eff : BYTE ;	//Phasenstrom L2 0..20 000 A [0..2 000 000]
   Strom_L2_Eff1 : BYTE ;
   Strom_L2_Eff2 : BYTE ;
   Strom_L2_Eff3 : BYTE ;
   Strom_L3_Eff : BYTE ;	//Phasenstrom L3 0..20 000 A [0..2 000 000]
   Strom_L3_Eff1 : BYTE ;
   Strom_L3_Eff2 : BYTE ;
   Strom_L3_Eff3 : BYTE ;
   U_Elektronik : BYTE ;	//Versorgungsspannung der Elektronik
   U_Elektronik1 : BYTE ;
   Kuehlkoerpertemp : BYTE ;	//Kühlkörpertemperatur
   Schaltelementerwaermung : BYTE ;	//Schaltelementerwärmung
   Rest_Abkuehlzeit : BYTE ;	//Verbleibende Abkülzeit des Schaltelementes
   Rest_Abkuehlzeit1 : BYTE ;
   T_Auslosereserve : BYTE ;	//Zeitliche Auslösereserve des thermischen Motormodells
   T_Auslosereserve1 : BYTE ;
   Ausgangsleistung : BYTE ;	//Ausgangsleistung 0..2 147 483 W [0.. 2 147 4830]
   Ausgangsleistung1 : BYTE ;
   Ausgangsleistung2 : BYTE ;
   Ausgangsleistung3 : BYTE ;
   Reserviert_13 : BYTE ;
   Reserviert_14 : BYTE ;
   Reserviert_15 : BYTE ;
   Reserviert_16 : BYTE ;
   Reserviert_17 : BYTE ;
   Reserviert_18 : BYTE ;
   Reserviert_19 : BYTE ;
   Reserviert_20 : BYTE ;
   Reserviert_21 : BYTE ;
   Reserviert_22 : BYTE ;
   Reserviert_23 : BYTE ;
   Reserviert_24 : BYTE ;
  END_STRUCT ;	
BEGIN
END_DATA_BLOCK

DATA_BLOCK "SWD-PKE"	// DB 31
AUTHOR : Simdon
FAMILY : PKE
NAME : PKE-2
VERSION : 0.1
  STRUCT
   Oil1 : UDT 31;
   Head_400 : UDT 31;
   Steering : UDT 31;
   Oil2 : UDT 31;
   Booster1 : UDT 31;
  END_STRUCT ;	
BEGIN
END_DATA_BLOCK

DATA_BLOCK "Daten-PKE"	// DB 32
AUTHOR : Simdon
FAMILY : PKE
NAME : PKE-3
VERSION : 0.1
  STRUCT
   PKE1_1 : REAL  := 3.000000e-001;
   PKE1_11 : REAL  := 3.300000e-001;
   PKE1_12 : REAL  := 3.600000e-001;
   PKE1_13 : REAL  := 4.000000e-001;
   PKE1_14 : REAL  := 4.300000e-001;
   PKE1_15 : REAL  := 4.700000e-001;
   PKE1_16 : REAL  := 5.000000e-001;
   PKE1_17 : REAL  := 5.600000e-001;
   PKE1_18 : REAL  := 6.300000e-001;
   PKE1_19 : REAL  := 7.000000e-001;
   PKE1_110 : REAL  := 7.700000e-001;
   PKE1_111 : REAL  := 8.300000e-001;
   PKE1_112 : REAL  := 9.000000e-001;
   PKE1_113 : REAL  := 1.000000e+000;
   PKE1_114 : REAL  := 1.100000e+000;
   PKE1_115 : REAL  := 1.200000e+000;
   PKE4_1 : REAL  := 1.000000e+000;
   PKE4_11 : REAL  := 1.100000e+000;
   PKE4_12 : REAL  := 1.200000e+000;
   PKE4_13 : REAL  := 1.300000e+000;
   PKE4_14 : REAL  := 1.420000e+000;
   PKE4_15 : REAL  := 1.550000e+000;
   PKE4_16 : REAL  := 1.700000e+000;
   PKE4_17 : REAL  := 1.900000e+000;
   PKE4_18 : REAL  := 2.100000e+000;
   PKE4_19 : REAL  := 2.400000e+000;
   PKE4_110 : REAL  := 2.600000e+000;
   PKE4_111 : REAL  := 2.800000e+000;
   PKE4_112 : REAL  := 3.000000e+000;
   PKE4_113 : REAL  := 3.300000e+000;
   PKE4_114 : REAL  := 3.700000e+000;
   PKE4_115 : REAL  := 4.000000e+000;
   PKE12_1 : REAL  := 3.000000e+000;
   PKE12_11 : REAL  := 3.300000e+000;
   PKE12_12 : REAL  := 3.600000e+000;
   PKE12_13 : REAL  := 4.000000e+000;
   PKE12_14 : REAL  := 4.300000e+000;
   PKE12_15 : REAL  := 4.700000e+000;
   PKE12_16 : REAL  := 5.000000e+000;
   PKE12_17 : REAL  := 5.600000e+000;
   PKE12_18 : REAL  := 6.300000e+000;
   PKE12_19 : REAL  := 7.000000e+000;
   PKE12_110 : REAL  := 7.700000e+000;
   PKE12_111 : REAL  := 8.300000e+000;
   PKE12_112 : REAL  := 9.000000e+000;
   PKE12_113 : REAL  := 1.000000e+001;
   PKE12_114 : REAL  := 1.100000e+001;
   PKE12_115 : REAL  := 1.200000e+001;
   PKE32_1 : REAL  := 8.000000e+000;
   PKE32_11 : REAL  := 8.800000e+000;
   PKE32_12 : REAL  := 9.700000e+000;
   PKE32_13 : REAL  := 1.050000e+001;
   PKE32_14 : REAL  := 1.150000e+001;
   PKE32_15 : REAL  := 1.250000e+001;
   PKE32_16 : REAL  := 1.350000e+001;
   PKE32_17 : REAL  := 1.500000e+001;
   PKE32_18 : REAL  := 1.700000e+001;
   PKE32_19 : REAL  := 1.900000e+001;
   PKE32_110 : REAL  := 2.050000e+001;
   PKE32_111 : REAL  := 2.200000e+001;
   PKE32_112 : REAL  := 2.400000e+001;
   PKE32_113 : REAL  := 2.700000e+001;
   PKE32_114 : REAL  := 2.900000e+001;
   PKE32_115 : REAL  := 3.200000e+001;
   PKE65_1 : REAL  := 1.600000e+001;
   PKE65_11 : REAL  := 1.760000e+001;
   PKE65_12 : REAL  := 1.930000e+001;
   PKE65_13 : REAL  := 2.130000e+001;
   PKE65_14 : REAL  := 2.300000e+001;
   PKE65_15 : REAL  := 2.480000e+001;
   PKE65_16 : REAL  := 2.680000e+001;
   PKE65_17 : REAL  := 3.000000e+001;
   PKE65_18 : REAL  := 3.360000e+001;
   PKE65_19 : REAL  := 3.770000e+001;
   PKE65_110 : REAL  := 4.090000e+001;
   PKE65_111 : REAL  := 4.440000e+001;
   PKE65_112 : REAL  := 4.810000e+001;
   PKE65_113 : REAL  := 5.330000e+001;
   PKE65_114 : REAL  := 5.860000e+001;
   PKE65_115 : REAL  := 6.500000e+001;
  END_STRUCT ;	
BEGIN
   PKE1_1 := 3.000000e-01;
   PKE1_11 := 3.300000e-01;
   PKE1_12 := 3.600000e-01;
   PKE1_13 := 4.000000e-01;
   PKE1_14 := 4.300000e-01;
   PKE1_15 := 4.700000e-01;
   PKE1_16 := 5.000000e-01;
   PKE1_17 := 5.600000e-01;
   PKE1_18 := 6.300000e-01;
   PKE1_19 := 7.000000e-01;
   PKE1_110 := 7.700000e-01;
   PKE1_111 := 8.300000e-01;
   PKE1_112 := 9.000000e-01;
   PKE1_113 := 1.000000e+00;
   PKE1_114 := 1.100000e+00;
   PKE1_115 := 1.200000e+00;
   PKE4_1 := 1.000000e+00;
   PKE4_11 := 1.100000e+00;
   PKE4_12 := 1.200000e+00;
   PKE4_13 := 1.300000e+00;
   PKE4_14 := 1.420000e+00;
   PKE4_15 := 1.550000e+00;
   PKE4_16 := 1.700000e+00;
   PKE4_17 := 1.900000e+00;
   PKE4_18 := 2.100000e+00;
   PKE4_19 := 2.400000e+00;
   PKE4_110 := 2.600000e+00;
   PKE4_111 := 2.800000e+00;
   PKE4_112 := 3.000000e+00;
   PKE4_113 := 3.300000e+00;
   PKE4_114 := 3.700000e+00;
   PKE4_115 := 4.000000e+00;
   PKE12_1 := 3.000000e+00;
   PKE12_11 := 3.300000e+00;
   PKE12_12 := 3.600000e+00;
   PKE12_13 := 4.000000e+00;
   PKE12_14 := 4.300000e+00;
   PKE12_15 := 4.700000e+00;
   PKE12_16 := 5.000000e+00;
   PKE12_17 := 5.600000e+00;
   PKE12_18 := 6.300000e+00;
   PKE12_19 := 7.000000e+00;
   PKE12_110 := 7.700000e+00;
   PKE12_111 := 8.300000e+00;
   PKE12_112 := 9.000000e+00;
   PKE12_113 := 1.000000e+01;
   PKE12_114 := 1.100000e+01;
   PKE12_115 := 1.200000e+01;
   PKE32_1 := 8.000000e+00;
   PKE32_11 := 8.800000e+00;
   PKE32_12 := 9.700000e+00;
   PKE32_13 := 1.050000e+01;
   PKE32_14 := 1.150000e+01;
   PKE32_15 := 1.250000e+01;
   PKE32_16 := 1.350000e+01;
   PKE32_17 := 1.500000e+01;
   PKE32_18 := 1.700000e+01;
   PKE32_19 := 1.900000e+01;
   PKE32_110 := 2.050000e+01;
   PKE32_111 := 2.200000e+01;
   PKE32_112 := 2.400000e+01;
   PKE32_113 := 2.700000e+01;
   PKE32_114 := 2.900000e+01;
   PKE32_115 := 3.200000e+01;
   PKE65_1 := 1.600000e+01;
   PKE65_11 := 1.760000e+01;
   PKE65_12 := 1.930000e+01;
   PKE65_13 := 2.130000e+01;
   PKE65_14 := 2.300000e+01;
   PKE65_15 := 2.480000e+01;
   PKE65_16 := 2.680000e+01;
   PKE65_17 := 3.000000e+01;
   PKE65_18 := 3.360000e+01;
   PKE65_19 := 3.770000e+01;
   PKE65_110 := 4.090000e+01;
   PKE65_111 := 4.440000e+01;
   PKE65_112 := 4.810000e+01;
   PKE65_113 := 5.330000e+01;
   PKE65_114 := 5.860000e+01;
   PKE65_115 := 6.500000e+01;
END_DATA_BLOCK

DATA_BLOCK "NZM"	// DB 33
VERSION : 0.1
  STRUCT
   x0 : BOOL ;
   x1 : BOOL ;
   x2 : BOOL ;
   x3 : BOOL ;
   x4 : BOOL ;
   x5 : BOOL ;
   x6 : BOOL ;
   x7 : BOOL ;
   NoIntCom : BOOL ;	//Interner Kommunikationsfehler
   Short : BOOL ;	//Kurzschluss Ausgang Q0 oder Q1
   S0_Error : BOOL ;	//Energiezähler ungültig
   OVLD2 : BOOL ;	//Überlastwarnung >120%
   DIAG : BOOL ;	//Sammeldiagnose
   Spare1 : BOOL ;
   PRSNT : BOOL ;	//Teilnehmer vorhanden
   Spare2 : BOOL ;
   POS1 : BOOL ;	//Position Leistungsschalter Bit 1
   Pos2 : BOOL ;	//Position Leistungsschalter Bit 2
   STAT1 : BOOL ;	//Status Leistungsschalter Bit 1
   STAT2 : BOOL ;	//Status Leistungsschalter Bit 2
   RDY : BOOL ;	//Einschaltbereit
   Spare3 : BOOL ;
   Spare4 : BOOL ;
   OVLD1 : BOOL ;	//Überlastwarnung >100%
   Spare5 : BOOL ;
   WARN : BOOL ;	//Sammelwarnung
   Spare6 : BOOL ;
   Spare7 : BOOL ;
   TRIP1 : BOOL ;	//Auslösegrund Bit 1
   TRIP2 : BOOL ;	//Auslösegrund Bit 2
   TRIP3 : BOOL ;	//Auslösegrund Bit 3
   OVLD0 : BOOL ;	//Lastwarnung >70%
   I_phase1 : INT ;	//Strom Phase L1
   I_Phase2 : INT ;	//Strom Phase L2
   I_Phase3 : INT ;	//Strom Phase L3
   I_Max : INT ;	//Gesamtstromaufnahme
  END_STRUCT ;	
BEGIN
END_DATA_BLOCK

DATA_BLOCK "DataLogging2"	// DB 57
TITLE = Eingelesene Werte der Gassensorik
AUTHOR : Simdon
FAMILY : Head
NAME : PC_Daten
VERSION : 0.1
  STRUCT
   Hum_HydrOil_PP : REAL ;	//Feuchtesensor Hydröl PPH
   PresFeedingline_PP : REAL ;	//Druck Speisekreis Container PP
   Returnlinefilter1_PP : REAL ;	//Rücklauffilter #1 Container-Aggregat
   Returnlinefilter2_PP : REAL ;	//Rücklauffilter #2 Container-Aggregat
   Bypassfilter_PP : REAL ;	//Bypassfilter Container-Aggregat
   Returnlinefilter_BK : REAL ;	//Rücklauffilter Bohrkopfaggregat
   Feedinglinefilter_BK : REAL ;	//Speisekreisfilter Bohrkopfaggregat
   Feedinglinefilter_PP : REAL ;	//Speisekreisfilter Power Pack Container
   PresFeedingline_BK : REAL ;	//Druck Speisekreis Bohrkopfaggregat
   Flowmeter_1_BK : REAL ;	//Durchfluß Kühlkreis #1 im Bohrkopf
   Flowmeter_2_BK : REAL ;	//Durchfluß Kühlkreis #2 im Bohrkopf
   Hum_HydrOil_BK : REAL ;	//Feuchtesensor Hydröl BKAG
   TempHead : REAL ;	//Umgebungstemperatur Bohrkopf
   Pres_CaseDrain : REAL ;	//Drucksensor Lecköl im Bohrkopf
   PresCaseDrain_BKAG : REAL ;	//Druck Lecköl im Bohrkopfaggregat
   Service_Hydr_PP : REAL ;	//Volumenstrom Hydraulikpumpe im Container-Hydraulikaggregat
   Spare : REAL ;
   Temp_Cool_EMotor : REAL ;	//Temperatur im Kühlkreis für den E-Motor im BKAG
   Temp_Cool_HydrOil : REAL ;	//Temperatur im Kühlkreis für das Hydr.Öl im BKAG
   P_Bento_BK : REAL ;	//Druck Bentonitzusatzkreis im Bohrkopf
   SlurryLine_In : REAL ;	//Druck Speiseleitung, Eingang am Bypass-Ventil
   Inter_8_Way : REAL ;	//Wegaufnehmer Dehnerstation 8 (BKAG)
   Inter_8_Force : REAL ;	//Kraft Dehnerstation 8 (BKAG)
   HD_Vol : REAL ;	//Durchfluss Wasserhochdrucksystem im Bohrkopf
   PresOut_EMotor : REAL ;	//Ausgangsdruck Kühlaggregat E-Motor BK
   Temp_CaseDrain : REAL ;	//Temperatur Lecköl
   Flow_CaseDrain : REAL ;	//Durchfluss Lecköl
  END_STRUCT ;	
BEGIN
END_DATA_BLOCK

DATA_BLOCK "Fault_DB"	// DB 58
TITLE = Ausgefallene Slaves und Hilfestellung für Container/Bohrkopfmot.
AUTHOR : Simdon
FAMILY : Fault
NAME : Fault_DB
VERSION : 0.1
  STRUCT
   Jacks_Start : BOOL ;	//Pressenmotor wurde gestartet
   JacksMot_Run : BOOL ;	//Pressenmotor läuft
   Fault_Steeringpump : BOOL ;	//Störung Steuerpumpe Container AG
   Fault_JackMot : BOOL ;	//Motorschutzschalter Pressenmotor
   Oillevel_PP : BOOL ;	//Ölstand im Container-AG
   Oiltemp_PP : BOOL ;	//Öltemperatur im Container-AG
   Cutter_Start : BOOL ;	//Bohrkopfmotor wurde gestartet
   Cutter_Run : BOOL ;	//Bohrkopfmotor läuft
   GeneralFault_SS : BOOL ;	//Sammelfehler Softstarter
   CommFault_SS : BOOL ;	//Kommunikationsfehler Softstarter
   Thermocoupler : BOOL ;	//Kaltleiter Bohrkopfmotor
   Oillevel_BK : BOOL ;	//Ölstand im Bohrkopf-AG
   Oiltemp_BK : BOOL ;	//Öltemperatur im Bohrkopf-AG
   CoolingMotor_BK : BOOL ;	//Störung Umwälzpumpe für Kühlkreis Bohrkopfmotor
   CoolingFlow_BK : BOOL ;	//Durchflussmenge für Kühlkreis Bohrkopfmotor zu gering
   Spare1 : BOOL ;
   Spare2 : BOOL ;
   Spare3 : BOOL ;
   DP_Dehner_1 : BOOL ;	//Slave Dehner 1
   DP_Dehner_2 : BOOL ;	//Slave Dehner 2
   DP_Dehner_3 : BOOL ;	//Slave Dehner 3
   DP_Pumpe_1 : BOOL ;	//Slave Spülpume 1 Sperrwaser
   DP_Pumpe_2 : BOOL ;	//Slave Spülpume 2 Sperrwaser
   DP_Sperrwasser : BOOL ;	//Slave Sperrwasserpumpe
   DP_ChargeFlow : BOOL ;	//Slave Flowmeter Chargeline
   DP_DischargeFlow : BOOL ;	//Slave Flowmeter Dischargeline
   DP_Chargepump : BOOL ;	//Slave FU Speisepumpe
   DP_Dischargepump : BOOL ;	//Slave FU Förderpumpe
   DP_Boosterpump1 : BOOL ;	//Slave FU Zusatzpumpe #1
   DP_Boosterpump2 : BOOL ;	//Slave FU Zusatzpumpe #2
   DP_PPH : BOOL ;	//Slave Hydraulikaggregat im Container
   DP_PPM : BOOL ;	//Slave Hauptschaltschrank
   DP_Pult_S : BOOL ;	//Slave Pult Smart Wire Darwin
   DP_Pult_T : BOOL ;	//Slave Pult Turck
   DP_BK_20 : BOOL ;	//Slave Piconet Bohrkopf Adr. 20
   DP_BK_21 : BOOL ;	//Slave Piconet Bohrkopf Adr. 21
   DP_BK_22 : BOOL ;	//Slave Piconet Bohrkopf Adr. 22
   DP_BK_23 : BOOL ;	//Slave Piconet Bohrkopf Adr. 23
   DP_BK_24 : BOOL ;	//Slave Piconet Bohrkopf Adr. 24
   DP_BK_25 : BOOL ;	//Slave Piconet Bohrkopf Adr. 25
   DP_BK_30 : BOOL ;	//Slave Piconet Bohrkopf Adr. 30
   DP_BKAG : BOOL ;	//Slave Bohrkopfaggregat
   DP_Dehner_4 : BOOL ;	//Slave Dehner 4
   DP_Dehner_5 : BOOL ;	//Slave Dehner 5
   DP_Dehner_6 : BOOL ;	//Slave Dehner 6
   DP_Cuttermotor : BOOL ;	//Slave Softstarter Schürfradmotor
   DP_HDPump : BOOL ;	//Salve HD-Pumpe
   DP_Bentonitpumpe : BOOL ;	//Slave Bentonitpumpe
  END_STRUCT ;	
BEGIN
END_DATA_BLOCK

DATA_BLOCK "Cyl_Force"	// DB 59
AUTHOR : Simdon
FAMILY : Head
NAME : CylForce
VERSION : 0.1
  STRUCT
   F_Cyl1 : REAL ;	//Kraft Steuerzylinder 1
   F_Cyl2 : REAL ;	//Kraft Steuerzylinder 2
   F_Cyl3 : REAL ;	//Kraft Steuerzylinder 3
   F_Cyl_All : REAL ;	//Kraft Steuerzylinder Gesamt
  END_STRUCT ;	
BEGIN
END_DATA_BLOCK

DATA_BLOCK "GLOBAL_DIAG_DB"	// DB 100
VERSION : 0.1
  STRUCT
   DATA_FIELD : ARRAY  [1 .. 50 ] OF //Interne Bearbeitung (nicht anwenderrelevant)
   BYTE ;
   SUM_SLAVES_DIAG : INT ;	//Anzahl der betroffenen Slaves (ausgefallen oder gestoert)
   LIST_SLAVES_NOT_PRESENT : ARRAY  [1 .. 4 ] OF //Liste der ausgefallenen Slaves
   DWORD ;
   LIST_SLAVES_ERROR : ARRAY  [1 .. 4 ] OF //Liste der gestoerten Slaves
   DWORD ;
   RETVAL : INT ;	//Fehlerinformation
   BUSY : BOOL ;	//Auswertung laeuft
  END_STRUCT ;	
BEGIN
END_DATA_BLOCK

DATA_BLOCK "Glaettung_DB"	// DB 101
AUTHOR : Simdon
FAMILY : Distance
NAME : GlaettDB
VERSION : 0.0
"Glaettung"
BEGIN
END_DATA_BLOCK

DATA_BLOCK "LV_Speed_DB"	// DB 102
AUTHOR : Simdon
FAMILY : Distance
NAME : Speed_LV
VERSION : 0.1
  STRUCT
   Diff_time_high : DINT ;	//Länge des Impulses in ms
   Diff_time_low : DINT ;	//Zeit zwischen den Impulsen in ms
   Diff_time : REAL ;	//Zeit von Impuls zu Impuls in ms
   Speed_LV : REAL ;	//Geschwindigkeit ohne Glättung
   SysTime : TIME ;	//Systemzeit in ms
   rStrecke : REAL ;	//aktuell zurückgelegte Strecke
   rStrecke_alt : REAL ;	//gemerkte zurückgelegte Strecke
   diTime_Stop : DINT ;	//Stopzeit für Messung merken
   diTime_Start : DINT ;	//Startzeit für Messung merken
   xAbfrage1 : BOOL ;	//Hilfsmerker für Geschwindigkeitsmessung
   xAbfrage2 : BOOL ;	//Hilfsmerker für Geschwindigkeitsmessung
   xStartzeit_Flanke : BOOL ;	//Flankenmerker für Geschwindigkeitsmessung
   xStartzeit_merken : BOOL ;	//Hilfsmerker für Geschwindigkeitsmessung
   xStopzeit_Flanke : BOOL ;	//Flankenmerker für Geschwindigkeitsmessung
   xStopzeit_merken : BOOL ;	//Hilfsmerker für Geschwindigkeitsmessung
  END_STRUCT ;	
BEGIN
END_DATA_BLOCK

DATA_BLOCK "DB-Altivar"	// DB 112
TITLE = Datenbaustein für Altivar 61 Umrichter
AUTHOR : Simdon
FAMILY : Motoren
NAME : DB_Altiv
VERSION : 0.1
  STRUCT
   Charge : UDT 112;
   Discharge : UDT 112;
   Booster1 : UDT 112;
   Booster2 : UDT 112;
  END_STRUCT ;	
BEGIN
   Charge.EA_Adr_1 := 488;
   Discharge.EA_Adr_1 := 508;
   Booster1.EA_Adr_1 := 528;
   Booster2.EA_Adr_1 := 548;
END_DATA_BLOCK

DATA_BLOCK "DETAIL_DIAG_DB"	// DB 125
VERSION : 0.0
"DETAIL_DP_DIAG"
BEGIN
END_DATA_BLOCK

DATA_BLOCK "D&T"	// DB 126
VERSION : 0.1
  STRUCT
   DT_Start : DATE_AND_TIME ;	//vorläufige Platzhaltervariable
   DT_Vergleich : DATE_AND_TIME ;
   DT_Aktuell : DATE_AND_TIME ;
   DT_1 : DATE_AND_TIME ;
   Vergleich : DWORD  := DW#16#15;
  END_STRUCT ;	
BEGIN
END_DATA_BLOCK

ORGANIZATION_BLOCK "MainControl"	// OB 1
TITLE = mts1000M2; Letzter Stand: 28.02.2019 NSI (Auslieferung)
VERSION : 0.1
VAR_TEMP
  TEMP0 : BYTE ;
  TEMP1 : BYTE ;
  TEMP2 : BYTE ;
  TEMP3 : BYTE ;
  TEMP4 : BYTE ;
  TEMP5 : BYTE ;
  TEMP6 : INT ;
  TEMP7 : INT ;
  TEMP8 : INT ;
  TEMP9 : DATE_AND_TIME ;
END_VAR
BEGIN
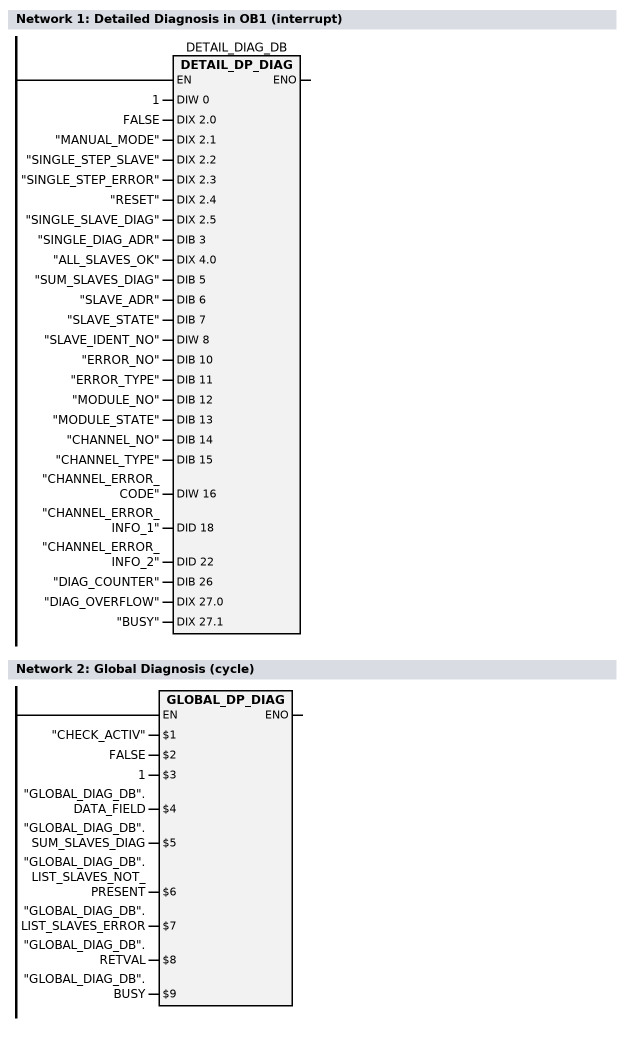
NETWORK
TITLE = Detailed Diagnosis in OB1 (interrupt)
      CALL  "DETAIL_DP_DIAG" , "DETAIL_DIAG_DB" (
           DIW 0                    := 1,
           DIX 2.0                  := FALSE,
           DIX 2.1                  := "MANUAL_MODE",
           DIX 2.2                  := "SINGLE_STEP_SLAVE",
           DIX 2.3                  := "SINGLE_STEP_ERROR",
           DIX 2.4                  := "RESET",
           DIX 2.5                  := "SINGLE_SLAVE_DIAG",
           DIB 3                    := "SINGLE_DIAG_ADR",
           DIX 4.0                  := "ALL_SLAVES_OK",
           DIB 5                    := "SUM_SLAVES_DIAG",
           DIB 6                    := "SLAVE_ADR",
           DIB 7                    := "SLAVE_STATE",
           DIW 8                    := "SLAVE_IDENT_NO",
           DIB 10                   := "ERROR_NO",
           DIB 11                   := "ERROR_TYPE",
           DIB 12                   := "MODULE_NO",
           DIB 13                   := "MODULE_STATE",
           DIB 14                   := "CHANNEL_NO",
           DIB 15                   := "CHANNEL_TYPE",
           DIW 16                   := "CHANNEL_ERROR_CODE",
           DID 18                   := "CHANNEL_ERROR_INFO_1",
           DID 22                   := "CHANNEL_ERROR_INFO_2",
           DIB 26                   := "DIAG_COUNTER",
           DIX 27.0                 := "DIAG_OVERFLOW",
           DIX 27.1                 := "BUSY");
NETWORK
TITLE = Global Diagnosis (cycle)
      CALL  "GLOBAL_DP_DIAG" (
           $1                       := "CHECK_ACTIV",
           $2                       := FALSE,
           $3                       := 1,
           $4                       := "GLOBAL_DIAG_DB".DATA_FIELD,
           $5                       := "GLOBAL_DIAG_DB".SUM_SLAVES_DIAG,
           $6                       := "GLOBAL_DIAG_DB".LIST_SLAVES_NOT_PRESENT,
           $7                       := "GLOBAL_DIAG_DB".LIST_SLAVES_ERROR,
           $8                       := "GLOBAL_DIAG_DB".RETVAL,
           $9                       := "GLOBAL_DIAG_DB".BUSY);
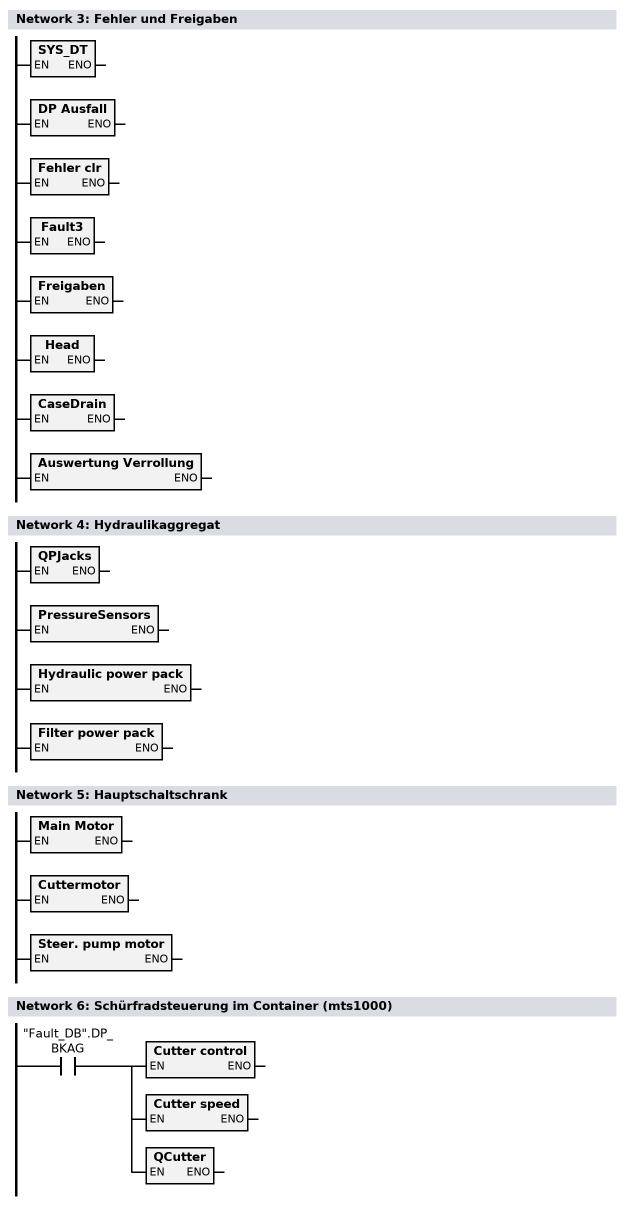
NETWORK
TITLE = Fehler und Freigaben
      CALL  "SYS_DT";
      CALL  "DP Ausfall";
      CALL  "Fehler clr";
      CALL  "Fault3";
      CALL  "Freigaben";
      CALL  "Head";
      CALL  "CaseDrain";
      CALL  "Auswertung Verrollung";
NETWORK
TITLE = Hydraulikaggregat
      CALL  "QPJacks";
      CALL  "PressureSensors";
      CALL  "Hydraulic power pack";
      CALL  "Filter power pack";
NETWORK
TITLE = Hauptschaltschrank
      CALL  "Main Motor";
      CALL  "Cuttermotor";
      CALL  "Steer. pump motor";
NETWORK
TITLE = Schürfradsteuerung im Container (mts1000)
      A     "Fault_DB".DP_BKAG;
      =     L 20.0;
      A     L 20.0;
      JNB   _001;
      CALL  "Cutter control";
_001: NOP   0;
      A     L 20.0;
      JNB   _002;
      CALL  "Cutter speed";
_002: NOP   0;
      A     L 20.0;
      JNB   _003;
      CALL  "QCutter";
_003: NOP   0;
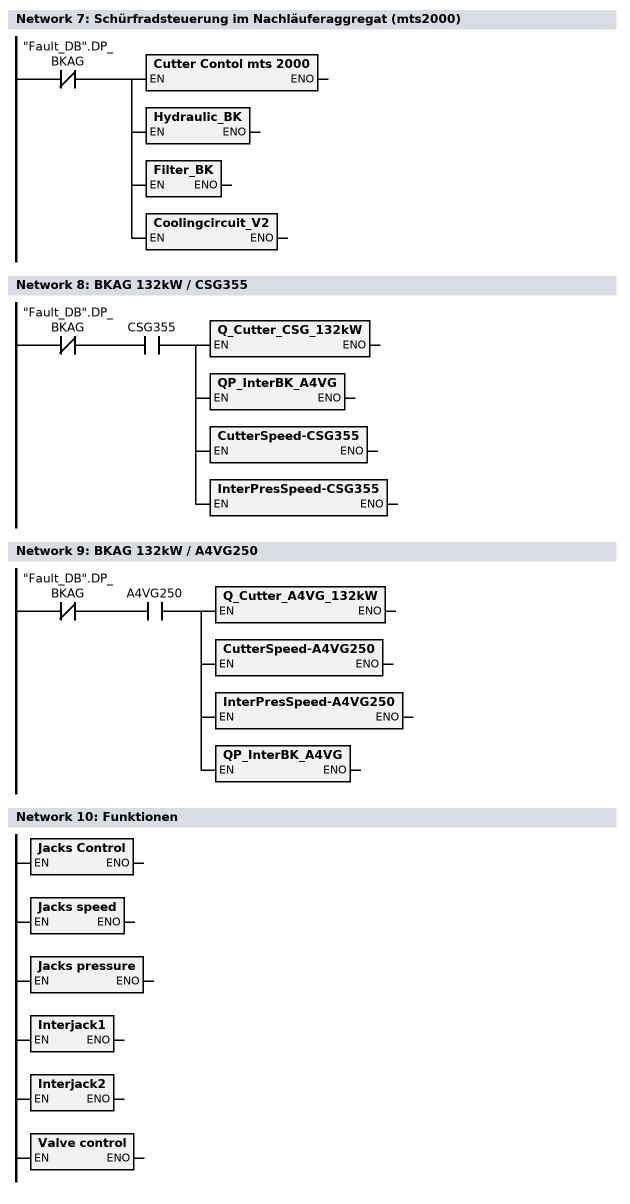
NETWORK
TITLE = Schürfradsteuerung im Nachläuferaggregat (mts2000)
      AN    "Fault_DB".DP_BKAG;
      =     L 20.0;
      A     L 20.0;
      JNB   _004;
      CALL  "Cutter Contol mts 2000";
_004: NOP   0;
      A     L 20.0;
      JNB   _005;
      CALL  "Hydraulic_BK";
_005: NOP   0;
      A     L 20.0;
      JNB   _006;
      CALL  "Filter_BK";
_006: NOP   0;
      A     L 20.0;
      JNB   _007;
      CALL  "Coolingcircuit_V2";
_007: NOP   0;
NETWORK
TITLE = BKAG 132kW / CSG355
      AN    "Fault_DB".DP_BKAG;
      A     "CSG355";
      =     L 20.0;
      A     L 20.0;
      JNB   _008;
      CALL  "Q_Cutter_CSG_132kW";
_008: NOP   0;
      A     L 20.0;
      JNB   _009;
      CALL  "QP_InterBK_A4VG";
_009: NOP   0;
      A     L 20.0;
      JNB   _00a;
      CALL  "CutterSpeed-CSG355";
_00a: NOP   0;
      A     L 20.0;
      JNB   _00b;
      CALL  "InterPresSpeed-CSG355";
_00b: NOP   0;
NETWORK
TITLE = BKAG 132kW / A4VG250
      AN    "Fault_DB".DP_BKAG;
      A     "A4VG250";
      =     L 20.0;
      A     L 20.0;
      JNB   _00c;
      CALL  "Q_Cutter_A4VG_132kW";
_00c: NOP   0;
      A     L 20.0;
      JNB   _00d;
      CALL  "CutterSpeed-A4VG250";
_00d: NOP   0;
      A     L 20.0;
      JNB   _00e;
      CALL  "InterPresSpeed-A4VG250";
_00e: NOP   0;
      A     L 20.0;
      JNB   _00f;
      CALL  "QP_InterBK_A4VG";
_00f: NOP   0;
NETWORK
TITLE = Funktionen
      CALL  "Jacks Control";
      CALL  "Jacks speed";
      CALL  "Jacks pressure";
      CALL  "Interjack1";
      CALL  "Interjack2";
      CALL  "Valve control";
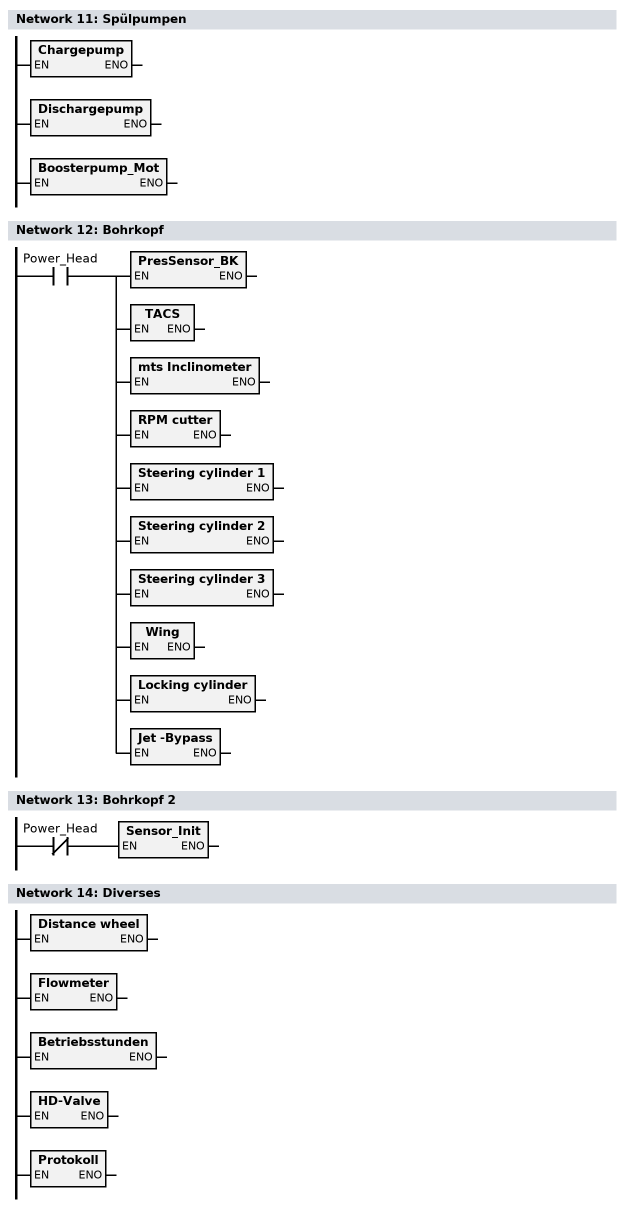
NETWORK
TITLE = Spülpumpen
      CALL  "Chargepump";
      CALL  "Dischargepump";
      CALL  "Boosterpump_Mot";
NETWORK
TITLE = Bohrkopf
      A     "Power_Head";
      =     L 20.0;
      A     L 20.0;
      JNB   _010;
      CALL  "PresSensor_BK";
_010: NOP   0;
      A     L 20.0;
      JNB   _011;
      CALL  "TACS";
_011: NOP   0;
      A     L 20.0;
      JNB   _012;
      CALL  "mts Inclinometer";
_012: NOP   0;
      A     L 20.0;
      JNB   _013;
      CALL  "RPM cutter";
_013: NOP   0;
      A     L 20.0;
      JNB   _014;
      CALL  "Steering cylinder 1";
_014: NOP   0;
      A     L 20.0;
      JNB   _015;
      CALL  "Steering cylinder 2";
_015: NOP   0;
      A     L 20.0;
      JNB   _016;
      CALL  "Steering cylinder 3";
_016: NOP   0;
      A     L 20.0;
      JNB   _017;
      CALL  "Wing";
_017: NOP   0;
      A     L 20.0;
      JNB   _018;
      CALL  "Locking cylinder";
_018: NOP   0;
      A     L 20.0;
      JNB   _019;
      CALL  "Jet -Bypass";
_019: NOP   0;
NETWORK
TITLE = Bohrkopf 2
      AN    "Power_Head";
      JNB   _01a;
      CALL  "Sensor_Init";
_01a: NOP   0;
NETWORK
TITLE = Diverses
      CALL  "Distance wheel";
      CALL  "Flowmeter";
      CALL  "Betriebsstunden";
      CALL  "HD-Valve";
      CALL  "Protokoll";
END_ORGANIZATION_BLOCK

ORGANIZATION_BLOCK "CYC_INT3"	// OB 33
TITLE = "Cyclic Interrupt"
VERSION : 0.1
VAR_TEMP
  OB32_EV_CLASS : BYTE ;	//Bits 0-3 = 1 (Coming event), Bits 4-7 = 1 (Event class 1)
  OB32_STRT_INF : BYTE ;	//16#33 (OB 32 has started)
  OB32_PRIORITY : BYTE ;	//Priority of OB Execution
  OB32_OB_NUMBR : BYTE ;	//32 (Organization block 32, OB32)
  OB32_RESERVED_1 : BYTE ;	//Reserved for system
  OB32_RESERVED_2 : BYTE ;	//Reserved for system
  OB32_PHS_OFFSET : INT ;	//Phase offset (integer, milliseconds)
  OB32_RESERVED_3 : INT ;	//Reserved for system
  OB32_EXC_FREQ : INT ;	//Frequency of execution (msec)
  OB32_DATE_TIME : DATE_AND_TIME ;	//Date and time OB32 started
END_VAR
BEGIN
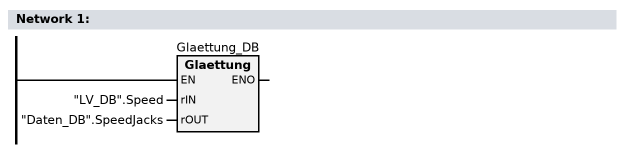
NETWORK
TITLE =
      CALL  "Glaettung" , "Glaettung_DB" (
           rIN                      := "LV_DB".Speed,
           rOUT                     := "Daten_DB".SpeedJacks);
      NOP   0;
END_ORGANIZATION_BLOCK

ORGANIZATION_BLOCK "I/O_FLT1"	// OB 82
VERSION : 0.1
VAR_TEMP
  OB82_EV_CLASS : BYTE ;	//16#39, Event class 3, Entering event state, Internal fault event
  OB82_FLT_ID : BYTE ;	//16#XX, Fault identifcation code
  OB82_PRIORITY : BYTE ;	//26/28 (Priority of 1 is lowest)
  OB82_OB_NUMBR : BYTE ;	//82 (Organization block 82, OB82)
  OB82_RESERVED_1 : BYTE ;	//Reserved for system
  OB82_IO_FLAG : BYTE ;	//Input (01010100), Output (01010101)
  OB82_MDL_ADDR : INT ;	//Base address of module with fault
  OB82_MDL_DEFECT : BOOL ;	//Module defective
  OB82_INT_FAULT : BOOL ;	//Internal fault
  OB82_EXT_FAULT : BOOL ;	//External fault
  OB82_PNT_INFO : BOOL ;	//Point information
  OB82_EXT_VOLTAGE : BOOL ;	//External voltage low
  OB82_FLD_CONNCTR : BOOL ;	//Field wiring connector missing
  OB82_NO_CONFIG : BOOL ;	//Module has no configuration data
  OB82_CONFIG_ERR : BOOL ;	//Module has configuration error
  OB82_MDL_TYPE : BYTE ;	//Type of module
  OB82_SUB_NDL_ERR : BOOL ;	//Sub-Module is missing or has error
  OB82_COMM_FAULT : BOOL ;	//Communication fault
  OB82_MDL_STOP : BOOL ;	//Module is stopped
  OB82_WTCH_DOG_FLT : BOOL ;	//Watch dog timer stopped module
  OB82_INT_PS_FLT : BOOL ;	//Internal power supply fault
  OB82_PRIM_BATT_FLT : BOOL ;	//Primary battery is in fault
  OB82_BCKUP_BATT_FLT : BOOL ;	//Backup battery is in fault
  OB82_RESERVED_2 : BOOL ;	//Reserved for system
  OB82_RACK_FLT : BOOL ;	//Rack fault, only for bus interface module
  OB82_PROC_FLT : BOOL ;	//Processor fault
  OB82_EPROM_FLT : BOOL ;	//EPROM fault
  OB82_RAM_FLT : BOOL ;	//RAM fault
  OB82_ADU_FLT : BOOL ;	//ADU fault
  OB82_FUSE_FLT : BOOL ;	//Fuse fault
  OB82_HW_INTR_FLT : BOOL ;	//Hardware interupt input in fault
  OB82_RESERVED_3 : BOOL ;	//Reserved for system
  OB82_DATE_TIME : DATE_AND_TIME ;	//Date and time OB82 started
END_VAR
BEGIN
NETWORK
TITLE = Detailed Diagnosis in OB82 (interrupt)
      CALL  "DETAIL_DP_DIAG" , "DETAIL_DIAG_DB" (
           DIW 0                    := 1,
           DIX 2.0                  := FALSE,
           DIX 2.1                  := "MANUAL_MODE",
           DIX 2.2                  := "SINGLE_STEP_SLAVE",
           DIX 2.3                  := "SINGLE_STEP_ERROR",
           DIX 2.4                  := "RESET",
           DIX 2.5                  := "SINGLE_SLAVE_DIAG",
           DIB 3                    := "SINGLE_DIAG_ADR",
           DIX 4.0                  := "ALL_SLAVES_OK",
           DIB 5                    := "SUM_SLAVES_DIAG",
           DIB 6                    := "SLAVE_ADR",
           DIB 7                    := "SLAVE_STATE",
           DIW 8                    := "SLAVE_IDENT_NO",
           DIB 10                   := "ERROR_NO",
           DIB 11                   := "ERROR_TYPE",
           DIB 12                   := "MODULE_NO",
           DIB 13                   := "MODULE_STATE",
           DIB 14                   := "CHANNEL_NO",
           DIB 15                   := "CHANNEL_TYPE",
           DIW 16                   := "CHANNEL_ERROR_CODE",
           DID 18                   := "CHANNEL_ERROR_INFO_1",
           DID 22                   := "CHANNEL_ERROR_INFO_2",
           DIB 26                   := "DIAG_COUNTER",
           DIX 27.0                 := "DIAG_OVERFLOW",
           DIX 27.1                 := "BUSY");
END_ORGANIZATION_BLOCK

ORGANIZATION_BLOCK "OBNL_FLT"	// OB 85
TITLE = "Organization Block (OB) Not Loaded Fault"
VERSION : 0.1
VAR_TEMP
  OB85_EV_CLASS : BYTE ;	//16#35 Event class 3
  OB85_FLT_ID : BYTE ;	//16#XX, Fault identification code
  OB85_PRIORITY : BYTE ;	//Priority of OB Execution
  OB85_OB_NUMBR : BYTE ;	//85 (Organization block 85, OB85)
  OB85_RESERVED_1 : BYTE ;	//Reserved for system
  OB85_RESERVED_2 : BYTE ;	//Reserved for system
  OB85_RESERVED_3 : INT ;	//Reserved for system
  OB85_ERR_EV_CLASS : BYTE ;	//Class of event causing error
  OB85_ERR_EV_NUM : BYTE ;	//Number of event causing error
  OB85_OB_PRIOR : BYTE ;	//Priority of OB causing error
  OB85_OB_NUM : BYTE ;	//Number of OB causing error
  OB85_DATE_TIME : DATE_AND_TIME ;	//Date and time OB85 started
END_VAR
BEGIN
// (block stored without names or comments; labels and parameter names are numbered)
END_ORGANIZATION_BLOCK

ORGANIZATION_BLOCK "RackFault"	// OB 86
VERSION : 0.1
VAR_TEMP
  OB86_EV_CLASS : BYTE ;	//16#38/39 Event class 3
  OB86_FLT_ID : BYTE ;	//16#C1/C4/C5, Fault identification code
  OB86_PRIORITY : BYTE ;	//26/28 (Priority of 1 is lowest)
  OB86_OB_NUMBR : BYTE ;	//86 (Organization block 86, OB86)
  OB86_RESERVED_1 : BYTE ;	//Reserved for system
  OB86_RESERVED_2 : BYTE ;	//Reserved for system
  OB86_MDL_ADDR : WORD ;	//Depending on fault identification code
  OB86_RACKS_FLTD : ARRAY  [0 .. 31 ] OF BOOL ;	//Racks in fault
  OB86_DATE_TIME : DATE_AND_TIME ;	//Date and time OB86 started
END_VAR
BEGIN
NETWORK
TITLE = Detailed Diagnosis in OB86 (interrupt)
      CALL  "DETAIL_DP_DIAG" , "DETAIL_DIAG_DB" (
           DIW 0                    := 1,
           DIX 2.0                  := FALSE,
           DIX 2.1                  := "MANUAL_MODE",
           DIX 2.2                  := "SINGLE_STEP_SLAVE",
           DIX 2.3                  := "SINGLE_STEP_ERROR",
           DIX 2.4                  := "RESET",
           DIX 2.5                  := "SINGLE_SLAVE_DIAG",
           DIB 3                    := "SINGLE_DIAG_ADR",
           DIX 4.0                  := "ALL_SLAVES_OK",
           DIB 5                    := "SUM_SLAVES_DIAG",
           DIB 6                    := "SLAVE_ADR",
           DIB 7                    := "SLAVE_STATE",
           DIW 8                    := "SLAVE_IDENT_NO",
           DIB 10                   := "ERROR_NO",
           DIB 11                   := "ERROR_TYPE",
           DIB 12                   := "MODULE_NO",
           DIB 13                   := "MODULE_STATE",
           DIB 14                   := "CHANNEL_NO",
           DIB 15                   := "CHANNEL_TYPE",
           DIW 16                   := "CHANNEL_ERROR_CODE",
           DID 18                   := "CHANNEL_ERROR_INFO_1",
           DID 22                   := "CHANNEL_ERROR_INFO_2",
           DIB 26                   := "DIAG_COUNTER",
           DIX 27.0                 := "DIAG_OVERFLOW",
           DIX 27.1                 := "BUSY");
END_ORGANIZATION_BLOCK

ORGANIZATION_BLOCK "COMPLETE RESTART"	// OB 100
TITLE = "Complete Restart"
VERSION : 0.1
VAR_TEMP
  OB100_EV_CLASS : BYTE ;	//16#13, Event class 1, Entering event state, Event logged in diagnostic buffer
  OB100_STRTUP : BYTE ;	//16#81/82/83/84 Method of startup
  OB100_PRIORITY : BYTE ;	//Priority of OB Execution
  OB100_OB_NUMBR : BYTE ;	//100 (Organization block 100, OB100)
  OB100_RESERVED_1 : BYTE ;	//Reserved for system
  OB100_RESERVED_2 : BYTE ;	//Reserved for system
  OB100_STOP : WORD ;	//Event that caused CPU to stop (16#4xxx)
  OB100_STRT_INFO : DWORD ;	//Information on how system started
  OB100_DATE_TIME : DATE_AND_TIME ;	//Date and time OB100 started
  DTIni : BOOL ;
  ReturnWrite : INT ;
END_VAR
BEGIN
NETWORK
TITLE = Frequenzumrichter und Softstarter ausschalten
      CLR;
      =     "FU_DB1".C_UmrichterStart;
      =     "FU_DB1".D_UmrichterStart;
      =     "FU_DB1".B_UmrichterStart;
      =     "FU_DB1".B2_UmrichterStart;
      =     "FU_DB1".BK_UmrichterStart;
NETWORK
TITLE = Pressenmotor
      CLR;
      =     "MainJackMot_K";
      =     "MainJackMot_Start";
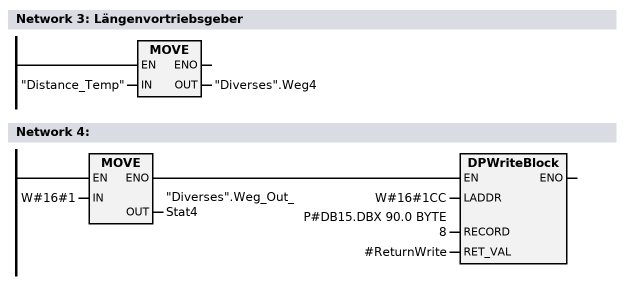
NETWORK
TITLE = Längenvortriebsgeber
      L     "Distance_Temp";
      T     "Diverses".Weg4;
NETWORK
TITLE =
      A(;
      L     W#16#1;
      T     "Diverses".Weg_Out_Stat4;
      SET;
      SAVE;
      CLR;
      A     BR;
      );
      JNB   _001;
      CALL  "DPWriteBlock" (
           LADDR                    := W#16#1CC,
           RECORD                   := P#DB15.DBX 90.0 BYTE 8,
           RET_VAL                  := #ReturnWrite);
_001: NOP   0;
END_ORGANIZATION_BLOCK

ORGANIZATION_BLOCK "PROG_ERR"	// OB 121
TITLE = "Programming Error"
VERSION : 0.1
VAR_TEMP
  OB121_EV_CLASS : BYTE ;	//16#25, Event class 2, Entering event state, Internal fault event
  OB121_SW_FLT : BYTE ;	//16#XX Software programming fault
  OB121_PRIORITY : BYTE ;	//Priority of OB Execution
  OB121_OB_NUMBR : BYTE ;	//121 (Organization block 121, OB121)
  OB121_BLK_TYPE : BYTE ;	//16#88/8A/8B/8C/8E Type of block fault occured in
  OB121_RESERVED_1 : BYTE ;	//Reserved for system
  OB121_FLT_REG : WORD ;	//16#XX Specific register that caused fault
  OB121_BLK_NUM : WORD ;	//Number of block that programming fault occured in
  OB121_PRG_ADDR : WORD ;	//Address in block where programming fault occured
  OB121_DATE_TIME : DATE_AND_TIME ;	//Date and time OB121 started
END_VAR
BEGIN
// (block stored without names or comments; labels and parameter names are numbered)
END_ORGANIZATION_BLOCK

ORGANIZATION_BLOCK "ModulError"	// OB 122
TITLE = "Module Access Error"
VERSION : 0.0
VAR_TEMP
  OB122_EV_CLASS : BYTE ;	//16#29, Event class 2, Entering event state, Internal fault event
  OB122_SW_FLT : BYTE ;	//16#XX Software error code
  OB122_PRIORITY : BYTE ;	//X = Priority of OB where fault occured (Priority of 1 is lowest)
  OB122_OB_NUMBR : BYTE ;	//122 (Organization block 122, OB122)
  OB122_BLK_TYPE : BYTE ;	//16#88/8A/8C/8E Type of block fault occured in
  OB122_MEM_AREA : BYTE ;	//Memory area where access error occured
  OB122_MEM_ADDR : WORD ;	//Memory address where access error occured
  OB122_BLK_NUM : WORD ;	//Block number in which error occured
  OB122_PRG_ADDR : WORD ;	//Program address where error occured
  OB122_DATE_TIME : DATE_AND_TIME ;	//Date and time OB1 started
END_VAR
BEGIN
NETWORK
TITLE =
END_ORGANIZATION_BLOCK
